	X =  165.960  mm,	Y =   -469.839  mm,	Z =   -309.000  mm,
	W =  90.000 deg,	P =   0.000 deg,	R =   90.000 deg
};
P[3008]{
   GP1:
	UF : 0, UT : 6,		CONFIG : 'N U T, 0, 0, 0',
	X =  164.763  mm,	Y =   -470.352  mm,	Z =   -309.000  mm,
	W =  90.000 deg,	P =   0.000 deg,	R =   90.000 deg
};
P[3009]{
   GP1:
	UF : 0, UT : 6,		CONFIG : 'N U T, 0, 0, 0',
	X =  163.654  mm,	Y =   -470.474  mm,	Z =   -309.000  mm,
	W =  90.000 deg,	P =   0.000 deg,	R =   90.000 deg
};
P[3010]{
   GP1:
	UF : 0, UT : 6,		CONFIG : 'N U T, 0, 0, 0',
	X =  163.001  mm,	Y =   -471.506  mm,	Z =   -309.100  mm,
	W =  90.000 deg,	P =   0.000 deg,	R =   90.000 deg
};
P[3011]{
   GP1:
	UF : 0, UT : 6,		CONFIG : 'N U T, 0, 0, 0',
	X =  162.078  mm,	Y =   -472.109  mm,	Z =   -309.100  mm,
	W =  90.000 deg,	P =   0.000 deg,	R =   90.000 deg
};
P[3012]{
   GP1:
	UF : 0, UT : 6,		CONFIG : 'N U T, 0, 0, 0',
	X =  161.118  mm,	Y =   -472.310  mm,	Z =   -309.000  mm,
	W =  90.000 deg,	P =   0.000 deg,	R =   90.000 deg
};
P[3013]{
   GP1:
	UF : 0, UT : 6,		CONFIG : 'N U T, 0, 0, 0',
	X =  160.747  mm,	Y =   -473.096  mm,	Z =   -309.000  mm,
	W =  90.000 deg,	P =   0.000 deg,	R =   90.000 deg
};
P[3014]{
   GP1:
	UF : 0, UT : 6,		CONFIG : 'N U T, 0, 0, 0',
	X =  159.614  mm,	Y =   -473.326  mm,	Z =   -312.206  mm,
	W =  90.000 deg,	P =   0.000 deg,	R =   90.000 deg
};
P[3015]{
   GP1:
	UF : 0, UT : 6,		CONFIG : 'N U T, 0, 0, 0',
	X =  158.718  mm,	Y =   -474.116  mm,	Z =   -309.000  mm,
	W =  90.000 deg,	P =   0.000 deg,	R =   90.000 deg
};
P[3016]{
   GP1:
	UF : 0, UT : 6,		CONFIG : 'N U T, 0, 0, 0',
	X =  157.157  mm,	Y =   -474.400  mm,	Z =   -309.000  mm,
	W =  90.000 deg,	P =   0.000 deg,	R =   90.000 deg
};
P[3017]{
   GP1:
	UF : 0, UT : 6,		CONFIG : 'N U T, 0, 0, 0',
	X =  156.715  mm,	Y =   -475.159  mm,	Z =   -320.034  mm,
	W =  90.000 deg,	P =   0.000 deg,	R =   90.000 deg
};
P[3018]{
   GP1:
	UF : 0, UT : 6,		CONFIG : 'N U T, 0, 0, 0',
	X =  155.908  mm,	Y =   -475.336  mm,	Z =   -309.000  mm,
	W =  90.000 deg,	P =   0.000 deg,	R =   90.000 deg
};
P[3019]{
   GP1:
	UF : 0, UT : 6,		CONFIG : 'N U T, 0, 0, 0',
	X =  154.941  mm,	Y =   -475.565  mm,	Z =   -309.000  mm,
	W =  90.000 deg,	P =   0.000 deg,	R =   90.000 deg
};
P[3020]{
   GP1:
	UF : 0, UT : 6,		CONFIG : 'N U T, 0, 0, 0',
	X =  154.314  mm,	Y =   -476.515  mm,	Z =   -309.000  mm,
	W =  90.000 deg,	P =   0.000 deg,	R =   90.000 deg
};
P[3021]{
   GP1:
	UF : 0, UT : 6,		CONFIG : 'N U T, 0, 0, 0',
	X =  153.381  mm,	Y =   -476.773  mm,	Z =   -309.000  mm,
	W =  90.000 deg,	P =   0.000 deg,	R =   90.000 deg
};
P[3022]{
   GP1:
	UF : 0, UT : 6,		CONFIG : 'N U T, 0, 0, 0',
	X =  161.189  mm,	Y =   -489.706  mm,	Z =   -309.000  mm,
	W =  90.000 deg,	P =   0.000 deg,	R =   90.000 deg
};
P[3023]{
   GP1:
	UF : 0, UT : 6,		CONFIG : 'N U T, 0, 0, 0',
	X =  162.232  mm,	Y =   -489.306  mm,	Z =   -309.000  mm,
	W =  90.000 deg,	P =   0.000 deg,	R =   90.000 deg
};
P[3024]{
   GP1:
	UF : 0, UT : 6,		CONFIG : 'N U T, 0, 0, 0',
	X =  162.974  mm,	Y =   -488.936  mm,	Z =   -309.000  mm,
	W =  90.000 deg,	P =   0.000 deg,	R =   90.000 deg
};
P[3025]{
   GP1:
	UF : 0, UT : 6,		CONFIG : 'N U T, 0, 0, 0',
	X =  164.233  mm,	Y =   -488.251  mm,	Z =   -309.000  mm,
	W =  90.000 deg,	P =   0.000 deg,	R =   90.000 deg
};
P[3026]{
   GP1:
	UF : 0, UT : 6,		CONFIG : 'N U T, 0, 0, 0',
	X =  166.230  mm,	Y =   -486.702  mm,	Z =   -309.000  mm,
	W =  90.000 deg,	P =   0.000 deg,	R =   90.000 deg
};
P[3027]{
   GP1:
	UF : 0, UT : 6,		CONFIG : 'N U T, 0, 0, 0',
	X =  167.168  mm,	Y =   -486.317  mm,	Z =   -309.000  mm,
	W =  90.000 deg,	P =   0.000 deg,	R =   90.000 deg
};
P[3028]{
   GP1:
	UF : 0, UT : 6,		CONFIG : 'N U T, 0, 0, 0',
	X =  167.771  mm,	Y =   -485.802  mm,	Z =   -309.000  mm,
	W =  90.000 deg,	P =   0.000 deg,	R =   90.000 deg
};
P[3029]{
   GP1:
	UF : 0, UT : 6,		CONFIG : 'N U T, 0, 0, 0',
	X =  168.725  mm,	Y =   -485.608  mm,	Z =   -309.000  mm,
	W =  90.000 deg,	P =   0.000 deg,	R =   90.000 deg
};
P[3030]{
   GP1:
	UF : 0, UT : 6,		CONFIG : 'N U T, 0, 0, 0',
	X =  170.097  mm,	Y =   -485.095  mm,	Z =   -309.000  mm,
	W =  90.000 deg,	P =   0.000 deg,	R =   90.000 deg
};
P[3031]{
   GP1:
	UF : 0, UT : 6,		CONFIG : 'N U T, 0, 0, 0',
	X =  171.086  mm,	Y =   -483.830  mm,	Z =   -310.570  mm,
	W =  90.000 deg,	P =   0.000 deg,	R =   90.000 deg
};
P[3032]{
   GP1:
	UF : 0, UT : 6,		CONFIG : 'N U T, 0, 0, 0',
	X =  172.239  mm,	Y =   -483.433  mm,	Z =   -309.100  mm,
	W =  90.000 deg,	P =   0.000 deg,	R =   90.000 deg
};
P[3033]{
   GP1:
	UF : 0, UT : 6,		CONFIG : 'N U T, 0, 0, 0',
	X =  173.577  mm,	Y =   -482.381  mm,	Z =   -309.100  mm,
	W =  90.000 deg,	P =   0.000 deg,	R =   90.000 deg
};
P[3034]{
   GP1:
	UF : 0, UT : 6,		CONFIG : 'N U T, 0, 0, 0',
	X =  174.632  mm,	Y =   -482.143  mm,	Z =   -316.236  mm,
	W =  90.000 deg,	P =   0.000 deg,	R =   90.000 deg
};
P[3035]{
   GP1:
	UF : 0, UT : 6,		CONFIG : 'N U T, 0, 0, 0',
	X =  176.654  mm,	Y =   -480.667  mm,	Z =   -309.100  mm,
	W =  90.000 deg,	P =   0.000 deg,	R =   90.000 deg
};
P[3036]{
   GP1:
	UF : 0, UT : 6,		CONFIG : 'N U T, 0, 0, 0',
	X =  178.148  mm,	Y =   -479.994  mm,	Z =   -309.100  mm,
	W =  90.000 deg,	P =   0.000 deg,	R =   90.000 deg
};
P[3037]{
   GP1:
	UF : 0, UT : 6,		CONFIG : 'N U T, 0, 0, 0',
	X =  179.964  mm,	Y =   -478.828  mm,	Z =   -309.000  mm,
	W =  90.000 deg,	P =   0.000 deg,	R =   90.000 deg
};
P[3038]{
   GP1:
	UF : 0, UT : 6,		CONFIG : 'N U T, 0, 0, 0',
	X =  181.856  mm,	Y =   -477.882  mm,	Z =   -309.000  mm,
	W =  90.000 deg,	P =   0.000 deg,	R =   90.000 deg
};
P[3039]{
   GP1:
	UF : 0, UT : 6,		CONFIG : 'N U T, 0, 0, 0',
	X =  182.674  mm,	Y =   -477.319  mm,	Z =   -309.000  mm,
	W =  90.000 deg,	P =   0.000 deg,	R =   90.000 deg
};
P[3040]{
   GP1:
	UF : 0, UT : 6,		CONFIG : 'N U T, 0, 0, 0',
	X =  183.656  mm,	Y =   -476.853  mm,	Z =   -309.000  mm,
	W =  90.000 deg,	P =   0.000 deg,	R =   90.000 deg
};
P[3041]{
   GP1:
	UF : 0, UT : 6,		CONFIG : 'N U T, 0, 0, 0',
	X =  185.064  mm,	Y =   -475.764  mm,	Z =   -309.100  mm,
	W =  90.000 deg,	P =   0.000 deg,	R =   90.000 deg
};
P[3042]{
   GP1:
	UF : 0, UT : 6,		CONFIG : 'N U T, 0, 0, 0',
	X =  186.024  mm,	Y =   -475.466  mm,	Z =   -309.000  mm,
	W =  90.000 deg,	P =   0.000 deg,	R =   90.000 deg
};
P[3043]{
   GP1:
	UF : 0, UT : 6,		CONFIG : 'N U T, 0, 0, 0',
	X =  186.459  mm,	Y =   -474.881  mm,	Z =   -309.000  mm,
	W =  90.000 deg,	P =   0.000 deg,	R =   90.000 deg
};
P[3044]{
   GP1:
	UF : 0, UT : 6,		CONFIG : 'N U T, 0, 0, 0',
	X =  187.871  mm,	Y =   -474.561  mm,	Z =   -309.000  mm,
	W =  90.000 deg,	P =   0.000 deg,	R =   90.000 deg
};
P[3045]{
   GP1:
	UF : 0, UT : 6,		CONFIG : 'N U T, 0, 0, 0',
	X =  189.558  mm,	Y =   -473.607  mm,	Z =   -309.000  mm,
	W =  90.000 deg,	P =   0.000 deg,	R =   90.000 deg
};
P[3046]{
   GP1:
	UF : 0, UT : 6,		CONFIG : 'N U T, 0, 0, 0',
	X =  190.537  mm,	Y =   -473.179  mm,	Z =   -309.100  mm,
	W =  90.000 deg,	P =   0.000 deg,	R =   90.000 deg
};
P[3047]{
   GP1:
	UF : 0, UT : 6,		CONFIG : 'N U T, 0, 0, 0',
	X =  190.960  mm,	Y =   -472.234  mm,	Z =   -309.000  mm,
	W =  90.000 deg,	P =   0.000 deg,	R =   90.000 deg
};
P[3048]{
   GP1:
	UF : 0, UT : 6,		CONFIG : 'N U T, 0, 0, 0',
	X =  193.639  mm,	Y =   -470.753  mm,	Z =   -309.000  mm,
	W =  90.000 deg,	P =   0.000 deg,	R =   90.000 deg
};
P[3049]{
   GP1:
	UF : 0, UT : 6,		CONFIG : 'N U T, 0, 0, 0',
	X =  195.285  mm,	Y =   -470.166  mm,	Z =   -309.000  mm,
	W =  90.000 deg,	P =   0.000 deg,	R =   90.000 deg
};
P[3050]{
   GP1:
	UF : 0, UT : 6,		CONFIG : 'N U T, 0, 0, 0',
	X =  196.338  mm,	Y =   -469.341  mm,	Z =   -312.108  mm,
	W =  90.000 deg,	P =   0.000 deg,	R =   90.000 deg
};
P[3051]{
   GP1:
	UF : 0, UT : 6,		CONFIG : 'N U T, 0, 0, 0',
	X =  197.381  mm,	Y =   -469.332  mm,	Z =   -326.194  mm,
	W =  90.000 deg,	P =   0.000 deg,	R =   90.000 deg
};
P[3052]{
   GP1:
	UF : 0, UT : 6,		CONFIG : 'N U T, 0, 0, 0',
	X =  197.799  mm,	Y =   -468.667  mm,	Z =   -320.599  mm,
	W =  90.000 deg,	P =   0.000 deg,	R =   90.000 deg
};
P[3053]{
   GP1:
	UF : 0, UT : 6,		CONFIG : 'N U T, 0, 0, 0',
	X =  199.838  mm,	Y =   -467.568  mm,	Z =   -309.000  mm,
	W =  90.000 deg,	P =   0.000 deg,	R =   90.000 deg
};
P[3054]{
   GP1:
	UF : 0, UT : 6,		CONFIG : 'N U T, 0, 0, 0',
	X =  200.850  mm,	Y =   -467.137  mm,	Z =   -309.000  mm,
	W =  90.000 deg,	P =   0.000 deg,	R =   90.000 deg
};
P[3055]{
   GP1:
	UF : 0, UT : 6,		CONFIG : 'N U T, 0, 0, 0',
	X =  201.586  mm,	Y =   -466.595  mm,	Z =   -309.100  mm,
	W =  90.000 deg,	P =   0.000 deg,	R =   90.000 deg
};
P[3056]{
   GP1:
	UF : 0, UT : 6,		CONFIG : 'N U T, 0, 0, 0',
	X =  202.447  mm,	Y =   -466.499  mm,	Z =   -316.149  mm,
	W =  90.000 deg,	P =   0.000 deg,	R =   90.000 deg
};
P[3057]{
   GP1:
	UF : 0, UT : 6,		CONFIG : 'N U T, 0, 0, 0',
	X =  203.353  mm,	Y =   -465.563  mm,	Z =   -319.247  mm,
	W =  90.000 deg,	P =   0.000 deg,	R =   90.000 deg
};
P[3058]{
   GP1:
	UF : 0, UT : 6,		CONFIG : 'N U T, 0, 0, 0',
	X =  204.948  mm,	Y =   -464.262  mm,	Z =   -309.000  mm,
	W =  90.000 deg,	P =   0.000 deg,	R =   90.000 deg
};
P[3059]{
   GP1:
	UF : 0, UT : 6,		CONFIG : 'N U T, 0, 0, 0',
	X =  206.055  mm,	Y =   -463.667  mm,	Z =   -309.000  mm,
	W =  90.000 deg,	P =   0.000 deg,	R =   90.000 deg
};
P[3060]{
   GP1:
	UF : 0, UT : 6,		CONFIG : 'N U T, 0, 0, 0',
	X =  206.857  mm,	Y =   -463.488  mm,	Z =   -309.000  mm,
	W =  90.000 deg,	P =   0.000 deg,	R =   90.000 deg
};
P[3061]{
   GP1:
	UF : 0, UT : 6,		CONFIG : 'N U T, 0, 0, 0',
	X =  207.561  mm,	Y =   -462.861  mm,	Z =   -309.000  mm,
	W =  90.000 deg,	P =   0.000 deg,	R =   90.000 deg
};
P[3062]{
   GP1:
	UF : 0, UT : 6,		CONFIG : 'N U T, 0, 0, 0',
	X =  208.392  mm,	Y =   -462.080  mm,	Z =   -309.100  mm,
	W =  90.000 deg,	P =   0.000 deg,	R =   90.000 deg
};
P[3063]{
   GP1:
	UF : 0, UT : 6,		CONFIG : 'N U T, 0, 0, 0',
	X =  209.725  mm,	Y =   -462.207  mm,	Z =   -324.192  mm,
	W =  90.000 deg,	P =   0.000 deg,	R =   90.000 deg
};
P[3064]{
   GP1:
	UF : 0, UT : 6,		CONFIG : 'N U T, 0, 0, 0',
	X =  210.434  mm,	Y =   -461.339  mm,	Z =   -309.000  mm,
	W =  90.000 deg,	P =   0.000 deg,	R =   90.000 deg
};
P[3065]{
   GP1:
	UF : 0, UT : 6,		CONFIG : 'N U T, 0, 0, 0',
	X =  211.216  mm,	Y =   -460.996  mm,	Z =   -318.087  mm,
	W =  90.000 deg,	P =   0.000 deg,	R =   90.000 deg
};
P[3066]{
   GP1:
	UF : 0, UT : 6,		CONFIG : 'N U T, 0, 0, 0',
	X =  211.856  mm,	Y =   -460.545  mm,	Z =   -309.000  mm,
	W =  90.000 deg,	P =   0.000 deg,	R =   90.000 deg
};
P[3067]{
   GP1:
	UF : 0, UT : 6,		CONFIG : 'N U T, 0, 0, 0',
	X =  213.067  mm,	Y =   -460.370  mm,	Z =   -316.222  mm,
	W =  90.000 deg,	P =   0.000 deg,	R =   90.000 deg
};
P[3068]{
   GP1:
	UF : 0, UT : 6,		CONFIG : 'N U T, 0, 0, 0',
	X =  213.309  mm,	Y =   -459.472  mm,	Z =   -309.100  mm,
	W =  90.000 deg,	P =   0.000 deg,	R =   90.000 deg
};
P[3069]{
   GP1:
	UF : 0, UT : 6,		CONFIG : 'N U T, 0, 0, 0',
	X =  214.258  mm,	Y =   -459.161  mm,	Z =   -323.141  mm,
	W =  90.000 deg,	P =   0.000 deg,	R =   90.000 deg
};
P[3070]{
   GP1:
	UF : 0, UT : 6,		CONFIG : 'N U T, 0, 0, 0',
	X =  215.681  mm,	Y =   -458.097  mm,	Z =   -320.747  mm,
	W =  90.000 deg,	P =   0.000 deg,	R =   90.000 deg
};
P[3071]{
   GP1:
	UF : 0, UT : 6,		CONFIG : 'N U T, 0, 0, 0',
	X =  216.597  mm,	Y =   -458.003  mm,	Z =   -310.970  mm,
	W =  90.000 deg,	P =   0.000 deg,	R =   90.000 deg
};
P[3072]{
   GP1:
	UF : 0, UT : 6,		CONFIG : 'N U T, 0, 0, 0',
	X =  217.463  mm,	Y =   -457.305  mm,	Z =   -319.124  mm,
	W =  90.000 deg,	P =   0.000 deg,	R =   90.000 deg
};
P[3073]{
   GP1:
	UF : 0, UT : 6,		CONFIG : 'N U T, 0, 0, 0',
	X =  218.185  mm,	Y =   -457.117  mm,	Z =   -309.000  mm,
	W =  90.000 deg,	P =   0.000 deg,	R =   90.000 deg
};
P[3074]{
   GP1:
	UF : 0, UT : 6,		CONFIG : 'N U T, 0, 0, 0',
	X =  219.140  mm,	Y =   -456.645  mm,	Z =   -319.283  mm,
	W =  90.000 deg,	P =   0.000 deg,	R =   90.000 deg
};
P[3075]{
   GP1:
	UF : 0, UT : 6,		CONFIG : 'N U T, 0, 0, 0',
	X =  219.698  mm,	Y =   -456.066  mm,	Z =   -309.000  mm,
	W =  90.000 deg,	P =   0.000 deg,	R =   90.000 deg
};
P[3076]{
   GP1:
	UF : 0, UT : 6,		CONFIG : 'N U T, 0, 0, 0',
	X =  220.893  mm,	Y =   -455.735  mm,	Z =   -325.142  mm,
	W =  90.000 deg,	P =   0.000 deg,	R =   90.000 deg
};
P[3077]{
   GP1:
	UF : 0, UT : 6,		CONFIG : 'N U T, 0, 0, 0',
	X =  221.443  mm,	Y =   -454.761  mm,	Z =   -309.000  mm,
	W =  90.000 deg,	P =   0.000 deg,	R =   90.000 deg
};
P[3078]{
   GP1:
	UF : 0, UT : 6,		CONFIG : 'N U T, 0, 0, 0',
	X =  222.869  mm,	Y =   -454.133  mm,	Z =   -309.000  mm,
	W =  90.000 deg,	P =   0.000 deg,	R =   90.000 deg
};
P[3079]{
   GP1:
	UF : 0, UT : 6,		CONFIG : 'N U T, 0, 0, 0',
	X =  223.946  mm,	Y =   -453.384  mm,	Z =   -309.000  mm,
	W =  90.000 deg,	P =   0.000 deg,	R =   90.000 deg
};
P[3080]{
   GP1:
	UF : 0, UT : 6,		CONFIG : 'N U T, 0, 0, 0',
	X =  225.188  mm,	Y =   -452.814  mm,	Z =   -309.100  mm,
	W =  90.000 deg,	P =   0.000 deg,	R =   90.000 deg
};
P[3081]{
   GP1:
	UF : 0, UT : 6,		CONFIG : 'N U T, 0, 0, 0',
	X =  226.063  mm,	Y =   -452.342  mm,	Z =   -309.000  mm,
	W =  90.000 deg,	P =   0.000 deg,	R =   90.000 deg
};
P[3082]{
   GP1:
	UF : 0, UT : 6,		CONFIG : 'N U T, 0, 0, 0',
	X =  227.719  mm,	Y =   -451.530  mm,	Z =   -309.000  mm,
	W =  90.000 deg,	P =   0.000 deg,	R =   90.000 deg
};
P[3083]{
   GP1:
	UF : 0, UT : 6,		CONFIG : 'N U T, 0, 0, 0',
	X =  228.471  mm,	Y =   -451.139  mm,	Z =   -309.100  mm,
	W =  90.000 deg,	P =   0.000 deg,	R =   90.000 deg
};
P[3084]{
   GP1:
	UF : 0, UT : 6,		CONFIG : 'N U T, 0, 0, 0',
	X =  229.322  mm,	Y =   -450.263  mm,	Z =   -309.100  mm,
	W =  90.000 deg,	P =   0.000 deg,	R =   90.000 deg
};
P[3085]{
   GP1:
	UF : 0, UT : 6,		CONFIG : 'N U T, 0, 0, 0',
	X =  230.058  mm,	Y =   -450.049  mm,	Z =   -309.100  mm,
	W =  90.000 deg,	P =   0.000 deg,	R =   90.000 deg
};
P[3086]{
   GP1:
	UF : 0, UT : 6,		CONFIG : 'N U T, 0, 0, 0',
	X =  231.335  mm,	Y =   -449.319  mm,	Z =   -309.100  mm,
	W =  90.000 deg,	P =   0.000 deg,	R =   90.000 deg
};
P[3087]{
   GP1:
	UF : 0, UT : 6,		CONFIG : 'N U T, 0, 0, 0',
	X =  232.003  mm,	Y =   -448.940  mm,	Z =   -309.000  mm,
	W =  90.000 deg,	P =   0.000 deg,	R =   90.000 deg
};
P[3088]{
   GP1:
	UF : 0, UT : 6,		CONFIG : 'N U T, 0, 0, 0',
	X =  233.065  mm,	Y =   -448.329  mm,	Z =   -309.000  mm,
	W =  90.000 deg,	P =   0.000 deg,	R =   90.000 deg
};
P[3089]{
   GP1:
	UF : 0, UT : 6,		CONFIG : 'N U T, 0, 0, 0',
	X =  234.366  mm,	Y =   -447.530  mm,	Z =   -309.000  mm,
	W =  90.000 deg,	P =   0.000 deg,	R =   90.000 deg
};
P[3090]{
   GP1:
	UF : 0, UT : 6,		CONFIG : 'N U T, 0, 0, 0',
	X =  235.449  mm,	Y =   -446.817  mm,	Z =   -309.000  mm,
	W =  90.000 deg,	P =   0.000 deg,	R =   90.000 deg
};
P[3091]{
   GP1:
	UF : 0, UT : 6,		CONFIG : 'N U T, 0, 0, 0',
	X =  237.066  mm,	Y =   -446.066  mm,	Z =   -309.000  mm,
	W =  90.000 deg,	P =   0.000 deg,	R =   90.000 deg
};
P[3092]{
   GP1:
	UF : 0, UT : 6,		CONFIG : 'N U T, 0, 0, 0',
	X =  237.996  mm,	Y =   -445.243  mm,	Z =   -309.100  mm,
	W =  90.000 deg,	P =   0.000 deg,	R =   90.000 deg
};
P[3093]{
   GP1:
	UF : 0, UT : 6,		CONFIG : 'N U T, 0, 0, 0',
	X =  239.589  mm,	Y =   -444.449  mm,	Z =   -309.000  mm,
	W =  90.000 deg,	P =   0.000 deg,	R =   90.000 deg
};
P[3094]{
   GP1:
	UF : 0, UT : 6,		CONFIG : 'N U T, 0, 0, 0',
	X =  240.520  mm,	Y =   -443.817  mm,	Z =   -309.100  mm,
	W =  90.000 deg,	P =   0.000 deg,	R =   90.000 deg
};
P[3095]{
   GP1:
	UF : 0, UT : 6,		CONFIG : 'N U T, 0, 0, 0',
	X =  241.814  mm,	Y =   -443.197  mm,	Z =   -309.000  mm,
	W =  90.000 deg,	P =   0.000 deg,	R =   90.000 deg
};
P[3096]{
   GP1:
	UF : 0, UT : 6,		CONFIG : 'N U T, 0, 0, 0',
	X =  242.713  mm,	Y =   -442.766  mm,	Z =   -309.100  mm,
	W =  90.000 deg,	P =   0.000 deg,	R =   90.000 deg
};
P[3097]{
   GP1:
	UF : 0, UT : 6,		CONFIG : 'N U T, 0, 0, 0',
	X =  244.190  mm,	Y =   -441.863  mm,	Z =   -309.000  mm,
	W =  90.000 deg,	P =   0.000 deg,	R =   90.000 deg
};
P[3098]{
   GP1:
	UF : 0, UT : 6,		CONFIG : 'N U T, 0, 0, 0',
	X =  245.074  mm,	Y =   -441.722  mm,	Z =   -309.000  mm,
	W =  90.000 deg,	P =   0.000 deg,	R =   90.000 deg
};
P[3099]{
   GP1:
	UF : 0, UT : 6,		CONFIG : 'N U T, 0, 0, 0',
	X =  245.736  mm,	Y =   -441.083  mm,	Z =   -309.000  mm,
	W =  90.000 deg,	P =   0.000 deg,	R =   90.000 deg
};
P[3100]{
   GP1:
	UF : 0, UT : 6,		CONFIG : 'N U T, 0, 0, 0',
	X =  246.253  mm,	Y =   -440.457  mm,	Z =   -327.144  mm,
	W =  90.000 deg,	P =   0.000 deg,	R =   90.000 deg
};
P[3101]{
   GP1:
	UF : 0, UT : 6,		CONFIG : 'N U T, 0, 0, 0',
	X =  247.353  mm,	Y =   -440.603  mm,	Z =   -309.000  mm,
	W =  90.000 deg,	P =   0.000 deg,	R =   90.000 deg
};
P[3102]{
   GP1:
	UF : 0, UT : 6,		CONFIG : 'N U T, 0, 0, 0',
	X =  248.262  mm,	Y =   -439.339  mm,	Z =   -309.000  mm,
	W =  90.000 deg,	P =   0.000 deg,	R =   90.000 deg
};
P[3103]{
   GP1:
	UF : 0, UT : 6,		CONFIG : 'N U T, 0, 0, 0',
	X =  249.447  mm,	Y =   -438.720  mm,	Z =   -311.305  mm,
	W =  90.000 deg,	P =   0.000 deg,	R =   90.000 deg
};
P[3104]{
   GP1:
	UF : 0, UT : 6,		CONFIG : 'N U T, 0, 0, 0',
	X =  249.968  mm,	Y =   -438.198  mm,	Z =   -309.000  mm,
	W =  90.000 deg,	P =   0.000 deg,	R =   90.000 deg
};
P[3105]{
   GP1:
	UF : 0, UT : 6,		CONFIG : 'N U T, 0, 0, 0',
	X =  250.759  mm,	Y =   -437.823  mm,	Z =   -309.000  mm,
	W =  90.000 deg,	P =   0.000 deg,	R =   90.000 deg
};
P[3106]{
   GP1:
	UF : 0, UT : 6,		CONFIG : 'N U T, 0, 0, 0',
	X =  251.597  mm,	Y =   -437.468  mm,	Z =   -309.000  mm,
	W =  90.000 deg,	P =   0.000 deg,	R =   90.000 deg
};
P[3107]{
   GP1:
	UF : 0, UT : 6,		CONFIG : 'N U T, 0, 0, 0',
	X =  252.430  mm,	Y =   -436.757  mm,	Z =   -309.100  mm,
	W =  90.000 deg,	P =   0.000 deg,	R =   90.000 deg
};
P[3108]{
   GP1:
	UF : 0, UT : 6,		CONFIG : 'N U T, 0, 0, 0',
	X =  254.468  mm,	Y =   -436.321  mm,	Z =   -323.840  mm,
	W =  90.000 deg,	P =   0.000 deg,	R =   90.000 deg
};
P[3109]{
   GP1:
	UF : 0, UT : 6,		CONFIG : 'N U T, 0, 0, 0',
	X =  256.029  mm,	Y =   -435.170  mm,	Z =   -311.041  mm,
	W =  90.000 deg,	P =   0.000 deg,	R =   90.000 deg
};
P[3110]{
   GP1:
	UF : 0, UT : 6,		CONFIG : 'N U T, 0, 0, 0',
	X =  257.288  mm,	Y =   -434.608  mm,	Z =   -309.000  mm,
	W =  90.000 deg,	P =   0.000 deg,	R =   90.000 deg
};
P[3111]{
   GP1:
	UF : 0, UT : 6,		CONFIG : 'N U T, 0, 0, 0',
	X =  258.792  mm,	Y =   -433.675  mm,	Z =   -309.000  mm,
	W =  90.000 deg,	P =   0.000 deg,	R =   90.000 deg
};
P[3112]{
   GP1:
	UF : 0, UT : 6,		CONFIG : 'N U T, 0, 0, 0',
	X =  259.578  mm,	Y =   -432.478  mm,	Z =   -309.000  mm,
	W =  90.000 deg,	P =   0.000 deg,	R =   90.000 deg
};
P[3113]{
   GP1:
	UF : 0, UT : 6,		CONFIG : 'N U T, 0, 0, 0',
	X =  260.631  mm,	Y =   -432.212  mm,	Z =   -309.050  mm,
	W =  90.000 deg,	P =   0.000 deg,	R =   90.000 deg
};
P[3114]{
   GP1:
	UF : 0, UT : 6,		CONFIG : 'N U T, 0, 0, 0',
	X =  262.213  mm,	Y =   -431.382  mm,	Z =   -309.000  mm,
	W =  90.000 deg,	P =   0.000 deg,	R =   90.000 deg
};
P[3115]{
   GP1:
	UF : 0, UT : 6,		CONFIG : 'N U T, 0, 0, 0',
	X =  263.149  mm,	Y =   -431.451  mm,	Z =   -309.100  mm,
	W =  90.000 deg,	P =   0.000 deg,	R =   90.000 deg
};
P[3116]{
   GP1:
	UF : 0, UT : 6,		CONFIG : 'N U T, 0, 0, 0',
	X =  264.028  mm,	Y =   -430.671  mm,	Z =   -309.100  mm,
	W =  90.000 deg,	P =   0.000 deg,	R =   90.000 deg
};
P[3117]{
   GP1:
	UF : 0, UT : 6,		CONFIG : 'N U T, 0, 0, 0',
	X =  264.974  mm,	Y =   -429.997  mm,	Z =   -309.100  mm,
	W =  90.000 deg,	P =   0.000 deg,	R =   90.000 deg
};
P[3118]{
   GP1:
	UF : 0, UT : 6,		CONFIG : 'N U T, 0, 0, 0',
	X =  265.683  mm,	Y =   -429.203  mm,	Z =   -309.000  mm,
	W =  90.000 deg,	P =   0.000 deg,	R =   90.000 deg
};
P[3119]{
   GP1:
	UF : 0, UT : 6,		CONFIG : 'N U T, 0, 0, 0',
	X =  266.507  mm,	Y =   -428.883  mm,	Z =   -309.000  mm,
	W =  90.000 deg,	P =   0.000 deg,	R =   90.000 deg
};
P[3120]{
   GP1:
	UF : 0, UT : 6,		CONFIG : 'N U T, 0, 0, 0',
	X =  266.981  mm,	Y =   -428.166  mm,	Z =   -309.000  mm,
	W =  90.000 deg,	P =   0.000 deg,	R =   90.000 deg
};
P[3121]{
   GP1:
	UF : 0, UT : 6,		CONFIG : 'N U T, 0, 0, 0',
	X =  267.993  mm,	Y =   -427.934  mm,	Z =   -309.000  mm,
	W =  90.000 deg,	P =   0.000 deg,	R =   90.000 deg
};
P[3122]{
   GP1:
	UF : 0, UT : 6,		CONFIG : 'N U T, 0, 0, 0',
	X =  269.454  mm,	Y =   -427.191  mm,	Z =   -309.000  mm,
	W =  90.000 deg,	P =   0.000 deg,	R =   90.000 deg
};
P[3123]{
   GP1:
	UF : 0, UT : 6,		CONFIG : 'N U T, 0, 0, 0',
	X =  270.364  mm,	Y =   -426.904  mm,	Z =   -309.100  mm,
	W =  90.000 deg,	P =   0.000 deg,	R =   90.000 deg
};
P[3124]{
   GP1:
	UF : 0, UT : 6,		CONFIG : 'N U T, 0, 0, 0',
	X =  271.038  mm,	Y =   -426.468  mm,	Z =   -309.000  mm,
	W =  90.000 deg,	P =   0.000 deg,	R =   90.000 deg
};
P[3125]{
   GP1:
	UF : 0, UT : 6,		CONFIG : 'N U T, 0, 0, 0',
	X =  272.037  mm,	Y =   -426.276  mm,	Z =   -309.000  mm,
	W =  90.000 deg,	P =   0.000 deg,	R =   90.000 deg
};
P[3126]{
   GP1:
	UF : 0, UT : 6,		CONFIG : 'N U T, 0, 0, 0',
	X =  272.459  mm,	Y =   -425.643  mm,	Z =   -324.061  mm,
	W =  90.000 deg,	P =   0.000 deg,	R =   90.000 deg
};
P[3127]{
   GP1:
	UF : 0, UT : 6,		CONFIG : 'N U T, 0, 0, 0',
	X =  273.163  mm,	Y =   -425.087  mm,	Z =   -309.000  mm,
	W =  90.000 deg,	P =   0.000 deg,	R =   90.000 deg
};
P[3128]{
   GP1:
	UF : 0, UT : 6,		CONFIG : 'N U T, 0, 0, 0',
	X =  274.713  mm,	Y =   -424.625  mm,	Z =   -322.101  mm,
	W =  90.000 deg,	P =   0.000 deg,	R =   90.000 deg
};
P[3129]{
   GP1:
	UF : 0, UT : 6,		CONFIG : 'N U T, 0, 0, 0',
	X =  275.243  mm,	Y =   -423.859  mm,	Z =   -309.000  mm,
	W =  90.000 deg,	P =   0.000 deg,	R =   90.000 deg
};
P[3130]{
   GP1:
	UF : 0, UT : 6,		CONFIG : 'N U T, 0, 0, 0',
	X =  276.293  mm,	Y =   -423.542  mm,	Z =   -309.000  mm,
	W =  90.000 deg,	P =   0.000 deg,	R =   90.000 deg
};
P[3131]{
   GP1:
	UF : 0, UT : 6,		CONFIG : 'N U T, 0, 0, 0',
	X =  276.935  mm,	Y =   -422.550  mm,	Z =   -309.000  mm,
	W =  90.000 deg,	P =   0.000 deg,	R =   90.000 deg
};
P[3132]{
   GP1:
	UF : 0, UT : 6,		CONFIG : 'N U T, 0, 0, 0',
	X =  277.995  mm,	Y =   -422.566  mm,	Z =   -309.100  mm,
	W =  90.000 deg,	P =   0.000 deg,	R =   90.000 deg
};
P[3133]{
   GP1:
	UF : 0, UT : 6,		CONFIG : 'N U T, 0, 0, 0',
	X =  279.606  mm,	Y =   -421.652  mm,	Z =   -309.100  mm,
	W =  90.000 deg,	P =   0.000 deg,	R =   90.000 deg
};
P[3134]{
   GP1:
	UF : 0, UT : 6,		CONFIG : 'N U T, 0, 0, 0',
	X =  280.174  mm,	Y =   -420.921  mm,	Z =   -309.000  mm,
	W =  90.000 deg,	P =   0.000 deg,	R =   90.000 deg
};
P[3135]{
   GP1:
	UF : 0, UT : 6,		CONFIG : 'N U T, 0, 0, 0',
	X =  280.833  mm,	Y =   -420.302  mm,	Z =   -309.000  mm,
	W =  90.000 deg,	P =   0.000 deg,	R =   90.000 deg
};
P[3136]{
   GP1:
	UF : 0, UT : 6,		CONFIG : 'N U T, 0, 0, 0',
	X =  281.961  mm,	Y =   -420.441  mm,	Z =   -309.000  mm,
	W =  90.000 deg,	P =   0.000 deg,	R =   90.000 deg
};
P[3137]{
   GP1:
	UF : 0, UT : 6,		CONFIG : 'N U T, 0, 0, 0',
	X =  282.907  mm,	Y =   -419.349  mm,	Z =   -309.000  mm,
	W =  90.000 deg,	P =   0.000 deg,	R =   90.000 deg
};
P[3138]{
   GP1:
	UF : 0, UT : 6,		CONFIG : 'N U T, 0, 0, 0',
	X =  284.593  mm,	Y =   -418.931  mm,	Z =   -312.196  mm,
	W =  90.000 deg,	P =   0.000 deg,	R =   90.000 deg
};
P[3139]{
   GP1:
	UF : 0, UT : 6,		CONFIG : 'N U T, 0, 0, 0',
	X =  285.638  mm,	Y =   -417.845  mm,	Z =   -309.000  mm,
	W =  90.000 deg,	P =   0.000 deg,	R =   90.000 deg
};
P[3140]{
   GP1:
	UF : 0, UT : 6,		CONFIG : 'N U T, 0, 0, 0',
	X =  287.168  mm,	Y =   -417.399  mm,	Z =   -309.000  mm,
	W =  90.000 deg,	P =   0.000 deg,	R =   90.000 deg
};
P[3141]{
   GP1:
	UF : 0, UT : 6,		CONFIG : 'N U T, 0, 0, 0',
	X =  288.074  mm,	Y =   -416.654  mm,	Z =   -309.000  mm,
	W =  90.000 deg,	P =   0.000 deg,	R =   90.000 deg
};
P[3142]{
   GP1:
	UF : 0, UT : 6,		CONFIG : 'N U T, 0, 0, 0',
	X =  288.701  mm,	Y =   -416.133  mm,	Z =   -309.000  mm,
	W =  90.000 deg,	P =   0.000 deg,	R =   90.000 deg
};
P[3143]{
   GP1:
	UF : 0, UT : 6,		CONFIG : 'N U T, 0, 0, 0',
	X =  289.901  mm,	Y =   -415.539  mm,	Z =   -309.000  mm,
	W =  90.000 deg,	P =   0.000 deg,	R =   90.000 deg
};
P[3144]{
   GP1:
	UF : 0, UT : 6,		CONFIG : 'N U T, 0, 0, 0',
	X =  290.454  mm,	Y =   -414.690  mm,	Z =   -309.100  mm,
	W =  90.000 deg,	P =   0.000 deg,	R =   90.000 deg
};
P[3145]{
   GP1:
	UF : 0, UT : 6,		CONFIG : 'N U T, 0, 0, 0',
	X =  291.404  mm,	Y =   -414.473  mm,	Z =   -309.000  mm,
	W =  90.000 deg,	P =   0.000 deg,	R =   90.000 deg
};
P[3146]{
   GP1:
	UF : 0, UT : 6,		CONFIG : 'N U T, 0, 0, 0',
	X =  293.101  mm,	Y =   -413.861  mm,	Z =   -309.000  mm,
	W =  90.000 deg,	P =   0.000 deg,	R =   90.000 deg
};
P[3147]{
   GP1:
	UF : 0, UT : 6,		CONFIG : 'N U T, 0, 0, 0',
	X =  294.183  mm,	Y =   -413.332  mm,	Z =   -309.100  mm,
	W =  90.000 deg,	P =   0.000 deg,	R =   90.000 deg
};
P[3148]{
   GP1:
	UF : 0, UT : 6,		CONFIG : 'N U T, 0, 0, 0',
	X =  295.158  mm,	Y =   -412.751  mm,	Z =   -309.000  mm,
	W =  90.000 deg,	P =   0.000 deg,	R =   90.000 deg
};
P[3149]{
   GP1:
	UF : 0, UT : 6,		CONFIG : 'N U T, 0, 0, 0',
	X =  296.044  mm,	Y =   -412.164  mm,	Z =   -309.000  mm,
	W =  90.000 deg,	P =   0.000 deg,	R =   90.000 deg
};
P[3150]{
   GP1:
	UF : 0, UT : 6,		CONFIG : 'N U T, 0, 0, 0',
	X =  296.655  mm,	Y =   -411.542  mm,	Z =   -309.100  mm,
	W =  90.000 deg,	P =   0.000 deg,	R =   90.000 deg
};
P[3151]{
   GP1:
	UF : 0, UT : 6,		CONFIG : 'N U T, 0, 0, 0',
	X =  297.891  mm,	Y =   -410.789  mm,	Z =   -309.100  mm,
	W =  90.000 deg,	P =   0.000 deg,	R =   90.000 deg
};
P[3152]{
   GP1:
	UF : 0, UT : 6,		CONFIG : 'N U T, 0, 0, 0',
	X =  298.854  mm,	Y =   -410.035  mm,	Z =   -309.000  mm,
	W =  90.000 deg,	P =   0.000 deg,	R =   90.000 deg
};
P[3153]{
   GP1:
	UF : 0, UT : 6,		CONFIG : 'N U T, 0, 0, 0',
	X =  299.668  mm,	Y =   -410.293  mm,	Z =   -309.100  mm,
	W =  90.000 deg,	P =   0.000 deg,	R =   90.000 deg
};
P[3154]{
   GP1:
	UF : 0, UT : 6,		CONFIG : 'N U T, 0, 0, 0',
	X =  299.957  mm,	Y =   -409.372  mm,	Z =   -309.100  mm,
	W =  90.000 deg,	P =   0.000 deg,	R =   90.000 deg
};
P[3155]{
   GP1:
	UF : 0, UT : 6,		CONFIG : 'N U T, 0, 0, 0',
	X =  301.093  mm,	Y =   -408.898  mm,	Z =   -320.865  mm,
	W =  90.000 deg,	P =   0.000 deg,	R =   90.000 deg
};
P[3156]{
   GP1:
	UF : 0, UT : 6,		CONFIG : 'N U T, 0, 0, 0',
	X =  302.572  mm,	Y =   -408.689  mm,	Z =   -309.000  mm,
	W =  90.000 deg,	P =   0.000 deg,	R =   90.000 deg
};
P[3157]{
   GP1:
	UF : 0, UT : 6,		CONFIG : 'N U T, 0, 0, 0',
	X =  302.970  mm,	Y =   -407.626  mm,	Z =   -309.000  mm,
	W =  90.000 deg,	P =   0.000 deg,	R =   90.000 deg
};
P[3158]{
   GP1:
	UF : 0, UT : 6,		CONFIG : 'N U T, 0, 0, 0',
	X =  303.741  mm,	Y =   -407.135  mm,	Z =   -309.000  mm,
	W =  90.000 deg,	P =   0.000 deg,	R =   90.000 deg
};
P[3159]{
   GP1:
	UF : 0, UT : 6,		CONFIG : 'N U T, 0, 0, 0',
	X =  304.855  mm,	Y =   -407.262  mm,	Z =   -309.100  mm,
	W =  90.000 deg,	P =   0.000 deg,	R =   90.000 deg
};
P[3160]{
   GP1:
	UF : 0, UT : 6,		CONFIG : 'N U T, 0, 0, 0',
	X =  305.478  mm,	Y =   -406.488  mm,	Z =   -309.000  mm,
	W =  90.000 deg,	P =   0.000 deg,	R =   90.000 deg
};
P[3161]{
   GP1:
	UF : 0, UT : 6,		CONFIG : 'N U T, 0, 0, 0',
	X =  307.123  mm,	Y =   -406.045  mm,	Z =   -309.100  mm,
	W =  90.000 deg,	P =   0.000 deg,	R =   90.000 deg
};
P[3162]{
   GP1:
	UF : 0, UT : 6,		CONFIG : 'N U T, 0, 0, 0',
	X =  307.854  mm,	Y =   -404.826  mm,	Z =   -309.033  mm,
	W =  90.000 deg,	P =   0.000 deg,	R =   90.000 deg
};
P[3163]{
   GP1:
	UF : 0, UT : 6,		CONFIG : 'N U T, 0, 0, 0',
	X =  309.131  mm,	Y =   -404.784  mm,	Z =   -309.100  mm,
	W =  90.000 deg,	P =   0.000 deg,	R =   90.000 deg
};
P[3164]{
   GP1:
	UF : 0, UT : 6,		CONFIG : 'N U T, 0, 0, 0',
	X =  309.845  mm,	Y =   -403.952  mm,	Z =   -309.100  mm,
	W =  90.000 deg,	P =   0.000 deg,	R =   90.000 deg
};
P[3165]{
   GP1:
	UF : 0, UT : 6,		CONFIG : 'N U T, 0, 0, 0',
	X =  310.858  mm,	Y =   -403.152  mm,	Z =   -309.000  mm,
	W =  90.000 deg,	P =   0.000 deg,	R =   90.000 deg
};
P[3166]{
   GP1:
	UF : 0, UT : 6,		CONFIG : 'N U T, 0, 0, 0',
	X =  311.586  mm,	Y =   -402.709  mm,	Z =   -309.000  mm,
	W =  90.000 deg,	P =   0.000 deg,	R =   90.000 deg
};
P[3167]{
   GP1:
	UF : 0, UT : 6,		CONFIG : 'N U T, 0, 0, 0',
	X =  312.311  mm,	Y =   -402.773  mm,	Z =   -309.000  mm,
	W =  90.000 deg,	P =   0.000 deg,	R =   90.000 deg
};
P[3168]{
   GP1:
	UF : 0, UT : 6,		CONFIG : 'N U T, 0, 0, 0',
	X =  313.053  mm,	Y =   -402.323  mm,	Z =   -309.100  mm,
	W =  90.000 deg,	P =   0.000 deg,	R =   90.000 deg
};
P[3169]{
   GP1:
	UF : 0, UT : 6,		CONFIG : 'N U T, 0, 0, 0',
	X =  314.188  mm,	Y =   -401.842  mm,	Z =   -309.100  mm,
	W =  90.000 deg,	P =   0.000 deg,	R =   90.000 deg
};
P[3170]{
   GP1:
	UF : 0, UT : 6,		CONFIG : 'N U T, 0, 0, 0',
	X =  314.964  mm,	Y =   -400.864  mm,	Z =   -309.000  mm,
	W =  90.000 deg,	P =   0.000 deg,	R =   90.000 deg
};
P[3171]{
   GP1:
	UF : 0, UT : 6,		CONFIG : 'N U T, 0, 0, 0',
	X =  315.588  mm,	Y =   -400.313  mm,	Z =   -309.000  mm,
	W =  90.000 deg,	P =   0.000 deg,	R =   90.000 deg
};
P[3172]{
   GP1:
	UF : 0, UT : 6,		CONFIG : 'N U T, 0, 0, 0',
	X =  316.389  mm,	Y =   -400.210  mm,	Z =   -309.000  mm,
	W =  90.000 deg,	P =   0.000 deg,	R =   90.000 deg
};
P[3173]{
   GP1:
	UF : 0, UT : 6,		CONFIG : 'N U T, 0, 0, 0',
	X =  317.487  mm,	Y =   -399.398  mm,	Z =   -309.000  mm,
	W =  90.000 deg,	P =   0.000 deg,	R =   90.000 deg
};
P[3174]{
   GP1:
	UF : 0, UT : 6,		CONFIG : 'N U T, 0, 0, 0',
	X =  318.789  mm,	Y =   -399.323  mm,	Z =   -309.000  mm,
	W =  90.000 deg,	P =   0.000 deg,	R =   90.000 deg
};
P[3175]{
   GP1:
	UF : 0, UT : 6,		CONFIG : 'N U T, 0, 0, 0',
	X =  318.884  mm,	Y =   -398.301  mm,	Z =   -309.000  mm,
	W =  90.000 deg,	P =   0.000 deg,	R =   90.000 deg
};
P[3176]{
   GP1:
	UF : 0, UT : 6,		CONFIG : 'N U T, 0, 0, 0',
	X =  320.086  mm,	Y =   -397.948  mm,	Z =   -309.000  mm,
	W =  90.000 deg,	P =   0.000 deg,	R =   90.000 deg
};
P[3177]{
   GP1:
	UF : 0, UT : 6,		CONFIG : 'N U T, 0, 0, 0',
	X =  321.476  mm,	Y =   -397.313  mm,	Z =   -309.100  mm,
	W =  90.000 deg,	P =   0.000 deg,	R =   90.000 deg
};
P[3178]{
   GP1:
	UF : 0, UT : 6,		CONFIG : 'N U T, 0, 0, 0',
	X =  323.081  mm,	Y =   -396.481  mm,	Z =   -309.000  mm,
	W =  90.000 deg,	P =   0.000 deg,	R =   90.000 deg
};
P[3179]{
   GP1:
	UF : 0, UT : 6,		CONFIG : 'N U T, 0, 0, 0',
	X =  324.212  mm,	Y =   -396.058  mm,	Z =   -309.100  mm,
	W =  90.000 deg,	P =   0.000 deg,	R =   90.000 deg
};
P[3180]{
   GP1:
	UF : 0, UT : 6,		CONFIG : 'N U T, 0, 0, 0',
	X =  324.493  mm,	Y =   -394.963  mm,	Z =   -309.100  mm,
	W =  90.000 deg,	P =   0.000 deg,	R =   90.000 deg
};
P[3181]{
   GP1:
	UF : 0, UT : 6,		CONFIG : 'N U T, 0, 0, 0',
	X =  325.264  mm,	Y =   -394.945  mm,	Z =   -309.100  mm,
	W =  90.000 deg,	P =   0.000 deg,	R =   90.000 deg
};
P[3182]{
   GP1:
	UF : 0, UT : 6,		CONFIG : 'N U T, 0, 0, 0',
	X =  326.233  mm,	Y =   -394.283  mm,	Z =   -309.100  mm,
	W =  90.000 deg,	P =   0.000 deg,	R =   90.000 deg
};
P[3183]{
   GP1:
	UF : 0, UT : 6,		CONFIG : 'N U T, 0, 0, 0',
	X =  327.626  mm,	Y =   -393.768  mm,	Z =   -309.000  mm,
	W =  90.000 deg,	P =   0.000 deg,	R =   90.000 deg
};
P[3184]{
   GP1:
	UF : 0, UT : 6,		CONFIG : 'N U T, 0, 0, 0',
	X =  329.137  mm,	Y =   -393.229  mm,	Z =   -309.000  mm,
	W =  90.000 deg,	P =   0.000 deg,	R =   90.000 deg
};
P[3185]{
   GP1:
	UF : 0, UT : 6,		CONFIG : 'N U T, 0, 0, 0',
	X =  329.591  mm,	Y =   -392.364  mm,	Z =   -309.000  mm,
	W =  90.000 deg,	P =   0.000 deg,	R =   90.000 deg
};
P[3186]{
   GP1:
	UF : 0, UT : 6,		CONFIG : 'N U T, 0, 0, 0',
	X =  330.664  mm,	Y =   -391.632  mm,	Z =   -309.000  mm,
	W =  90.000 deg,	P =   0.000 deg,	R =   90.000 deg
};
P[3187]{
   GP1:
	UF : 0, UT : 6,		CONFIG : 'N U T, 0, 0, 0',
	X =  331.564  mm,	Y =   -391.624  mm,	Z =   -309.000  mm,
	W =  90.000 deg,	P =   0.000 deg,	R =   90.000 deg
};
P[3188]{
   GP1:
	UF : 0, UT : 6,		CONFIG : 'N U T, 0, 0, 0',
	X =  332.310  mm,	Y =   -390.786  mm,	Z =   -325.993  mm,
	W =  90.000 deg,	P =   0.000 deg,	R =   90.000 deg
};
P[3189]{
   GP1:
	UF : 0, UT : 6,		CONFIG : 'N U T, 0, 0, 0',
	X =  333.203  mm,	Y =   -390.899  mm,	Z =   -309.000  mm,
	W =  90.000 deg,	P =   0.000 deg,	R =   90.000 deg
};
P[3190]{
   GP1:
	UF : 0, UT : 6,		CONFIG : 'N U T, 0, 0, 0',
	X =  333.996  mm,	Y =   -390.169  mm,	Z =   -309.000  mm,
	W =  90.000 deg,	P =   0.000 deg,	R =   90.000 deg
};
P[3191]{
   GP1:
	UF : 0, UT : 6,		CONFIG : 'N U T, 0, 0, 0',
	X =  341.415  mm,	Y =   -403.266  mm,	Z =   -309.100  mm,
	W =  90.000 deg,	P =   0.000 deg,	R =   90.000 deg
};
P[3192]{
   GP1:
	UF : 0, UT : 6,		CONFIG : 'N U T, 0, 0, 0',
	X =  340.535  mm,	Y =   -403.069  mm,	Z =   -309.000  mm,
	W =  90.000 deg,	P =   0.000 deg,	R =   90.000 deg
};
P[3193]{
   GP1:
	UF : 0, UT : 6,		CONFIG : 'N U T, 0, 0, 0',
	X =  340.148  mm,	Y =   -403.881  mm,	Z =   -309.000  mm,
	W =  90.000 deg,	P =   0.000 deg,	R =   90.000 deg
};
P[3194]{
   GP1:
	UF : 0, UT : 6,		CONFIG : 'N U T, 0, 0, 0',
	X =  339.227  mm,	Y =   -404.232  mm,	Z =   -309.000  mm,
	W =  90.000 deg,	P =   0.000 deg,	R =   90.000 deg
};
P[3195]{
   GP1:
	UF : 0, UT : 6,		CONFIG : 'N U T, 0, 0, 0',
	X =  338.194  mm,	Y =   -404.645  mm,	Z =   -311.898  mm,
	W =  90.000 deg,	P =   0.000 deg,	R =   90.000 deg
};
P[3196]{
   GP1:
	UF : 0, UT : 6,		CONFIG : 'N U T, 0, 0, 0',
	X =  337.156  mm,	Y =   -405.173  mm,	Z =   -309.100  mm,
	W =  90.000 deg,	P =   0.000 deg,	R =   90.000 deg
};
P[3197]{
   GP1:
	UF : 0, UT : 6,		CONFIG : 'N U T, 0, 0, 0',
	X =  335.370  mm,	Y =   -406.482  mm,	Z =   -309.000  mm,
	W =  90.000 deg,	P =   0.000 deg,	R =   90.000 deg
};
P[3198]{
   GP1:
	UF : 0, UT : 6,		CONFIG : 'N U T, 0, 0, 0',
	X =  334.478  mm,	Y =   -407.273  mm,	Z =   -309.100  mm,
	W =  90.000 deg,	P =   0.000 deg,	R =   90.000 deg
};
P[3199]{
   GP1:
	UF : 0, UT : 6,		CONFIG : 'N U T, 0, 0, 0',
	X =  333.604  mm,	Y =   -407.675  mm,	Z =   -309.000  mm,
	W =  90.000 deg,	P =   0.000 deg,	R =   90.000 deg
};
P[3200]{
   GP1:
	UF : 0, UT : 6,		CONFIG : 'N U T, 0, 0, 0',
	X =  332.753  mm,	Y =   -407.650  mm,	Z =   -309.000  mm,
	W =  90.000 deg,	P =   0.000 deg,	R =   90.000 deg
};
P[3201]{
   GP1:
	UF : 0, UT : 6,		CONFIG : 'N U T, 0, 0, 0',
	X =  331.874  mm,	Y =   -408.861  mm,	Z =   -309.100  mm,
	W =  90.000 deg,	P =   0.000 deg,	R =   90.000 deg
};
P[3202]{
   GP1:
	UF : 0, UT : 6,		CONFIG : 'N U T, 0, 0, 0',
	X =  331.186  mm,	Y =   -409.115  mm,	Z =   -309.000  mm,
	W =  90.000 deg,	P =   0.000 deg,	R =   90.000 deg
};
P[3203]{
   GP1:
	UF : 0, UT : 6,		CONFIG : 'N U T, 0, 0, 0',
	X =  330.283  mm,	Y =   -409.596  mm,	Z =   -309.100  mm,
	W =  90.000 deg,	P =   0.000 deg,	R =   90.000 deg
};
P[3204]{
   GP1:
	UF : 0, UT : 6,		CONFIG : 'N U T, 0, 0, 0',
	X =  329.083  mm,	Y =   -409.874  mm,	Z =   -315.562  mm,
	W =  90.000 deg,	P =   0.000 deg,	R =   90.000 deg
};
P[3205]{
   GP1:
	UF : 0, UT : 6,		CONFIG : 'N U T, 0, 0, 0',
	X =  327.493  mm,	Y =   -411.124  mm,	Z =   -309.000  mm,
	W =  90.000 deg,	P =   0.000 deg,	R =   90.000 deg
};
P[3206]{
   GP1:
	UF : 0, UT : 6,		CONFIG : 'N U T, 0, 0, 0',
	X =  326.758  mm,	Y =   -411.333  mm,	Z =   -309.000  mm,
	W =  90.000 deg,	P =   0.000 deg,	R =   90.000 deg
};
P[3207]{
   GP1:
	UF : 0, UT : 6,		CONFIG : 'N U T, 0, 0, 0',
	X =  326.458  mm,	Y =   -412.093  mm,	Z =   -309.000  mm,
	W =  90.000 deg,	P =   0.000 deg,	R =   90.000 deg
};
P[3208]{
   GP1:
	UF : 0, UT : 6,		CONFIG : 'N U T, 0, 0, 0',
	X =  325.294  mm,	Y =   -412.080  mm,	Z =   -309.000  mm,
	W =  90.000 deg,	P =   0.000 deg,	R =   90.000 deg
};
P[3209]{
   GP1:
	UF : 0, UT : 6,		CONFIG : 'N U T, 0, 0, 0',
	X =  324.335  mm,	Y =   -412.714  mm,	Z =   -309.000  mm,
	W =  90.000 deg,	P =   0.000 deg,	R =   90.000 deg
};
P[3210]{
   GP1:
	UF : 0, UT : 6,		CONFIG : 'N U T, 0, 0, 0',
	X =  323.397  mm,	Y =   -413.417  mm,	Z =   -309.100  mm,
	W =  90.000 deg,	P =   0.000 deg,	R =   90.000 deg
};
P[3211]{
   GP1:
	UF : 0, UT : 6,		CONFIG : 'N U T, 0, 0, 0',
	X =  322.140  mm,	Y =   -413.712  mm,	Z =   -309.000  mm,
	W =  90.000 deg,	P =   0.000 deg,	R =   90.000 deg
};
P[3212]{
   GP1:
	UF : 0, UT : 6,		CONFIG : 'N U T, 0, 0, 0',
	X =  321.655  mm,	Y =   -414.561  mm,	Z =   -309.100  mm,
	W =  90.000 deg,	P =   0.000 deg,	R =   90.000 deg
};
P[3213]{
   GP1:
	UF : 0, UT : 6,		CONFIG : 'N U T, 0, 0, 0',
	X =  321.152  mm,	Y =   -415.123  mm,	Z =   -309.201  mm,
	W =  90.000 deg,	P =   0.000 deg,	R =   90.000 deg
};
P[3214]{
   GP1:
	UF : 0, UT : 6,		CONFIG : 'N U T, 0, 0, 0',
	X =  319.716  mm,	Y =   -415.965  mm,	Z =   -309.000  mm,
	W =  90.000 deg,	P =   0.000 deg,	R =   90.000 deg
};
P[3215]{
   GP1:
	UF : 0, UT : 6,		CONFIG : 'N U T, 0, 0, 0',
	X =  318.873  mm,	Y =   -416.428  mm,	Z =   -309.000  mm,
	W =  90.000 deg,	P =   0.000 deg,	R =   90.000 deg
};
P[3216]{
   GP1:
	UF : 0, UT : 6,		CONFIG : 'N U T, 0, 0, 0',
	X =  317.083  mm,	Y =   -417.008  mm,	Z =   -309.000  mm,
	W =  90.000 deg,	P =   0.000 deg,	R =   90.000 deg
};
P[3217]{
   GP1:
	UF : 0, UT : 6,		CONFIG : 'N U T, 0, 0, 0',
	X =  316.060  mm,	Y =   -417.441  mm,	Z =   -309.100  mm,
	W =  90.000 deg,	P =   0.000 deg,	R =   90.000 deg
};
P[3218]{
   GP1:
	UF : 0, UT : 6,		CONFIG : 'N U T, 0, 0, 0',
	X =  315.602  mm,	Y =   -418.081  mm,	Z =   -309.100  mm,
	W =  90.000 deg,	P =   0.000 deg,	R =   90.000 deg
};
P[3219]{
   GP1:
	UF : 0, UT : 6,		CONFIG : 'N U T, 0, 0, 0',
	X =  314.664  mm,	Y =   -418.077  mm,	Z =   -309.000  mm,
	W =  90.000 deg,	P =   0.000 deg,	R =   90.000 deg
};
P[3220]{
   GP1:
	UF : 0, UT : 6,		CONFIG : 'N U T, 0, 0, 0',
	X =  313.962  mm,	Y =   -418.771  mm,	Z =   -309.000  mm,
	W =  90.000 deg,	P =   0.000 deg,	R =   90.000 deg
};
P[3221]{
   GP1:
	UF : 0, UT : 6,		CONFIG : 'N U T, 0, 0, 0',
	X =  313.017  mm,	Y =   -419.861  mm,	Z =   -311.050  mm,
	W =  90.000 deg,	P =   0.000 deg,	R =   90.000 deg
};
P[3222]{
   GP1:
	UF : 0, UT : 6,		CONFIG : 'N U T, 0, 0, 0',
	X =  312.425  mm,	Y =   -420.081  mm,	Z =   -309.000  mm,
	W =  90.000 deg,	P =   0.000 deg,	R =   90.000 deg
};
P[3223]{
   GP1:
	UF : 0, UT : 6,		CONFIG : 'N U T, 0, 0, 0',
	X =  312.258  mm,	Y =   -419.950  mm,	Z =   -309.100  mm,
	W =  90.000 deg,	P =   0.000 deg,	R =   90.000 deg
};
P[3224]{
   GP1:
	UF : 0, UT : 6,		CONFIG : 'N U T, 0, 0, 0',
	X =  311.923  mm,	Y =   -420.063  mm,	Z =   -309.000  mm,
	W =  90.000 deg,	P =   0.000 deg,	R =   90.000 deg
};
P[3225]{
   GP1:
	UF : 0, UT : 6,		CONFIG : 'N U T, 0, 0, 0',
	X =  311.627  mm,	Y =   -420.173  mm,	Z =   -309.000  mm,
	W =  90.000 deg,	P =   0.000 deg,	R =   90.000 deg
};
P[3226]{
   GP1:
	UF : 0, UT : 6,		CONFIG : 'N U T, 0, 0, 0',
	X =  311.468  mm,	Y =   -420.529  mm,	Z =   -309.100  mm,
	W =  90.000 deg,	P =   0.000 deg,	R =   90.000 deg
};
P[3227]{
   GP1:
	UF : 0, UT : 6,		CONFIG : 'N U T, 0, 0, 0',
	X =  311.355  mm,	Y =   -420.385  mm,	Z =   -309.000  mm,
	W =  90.000 deg,	P =   0.000 deg,	R =   90.000 deg
};
P[3228]{
   GP1:
	UF : 0, UT : 6,		CONFIG : 'N U T, 0, 0, 0',
	X =  311.189  mm,	Y =   -420.110  mm,	Z =   -309.000  mm,
	W =  90.000 deg,	P =   0.000 deg,	R =   90.000 deg
};
P[3229]{
   GP1:
	UF : 0, UT : 6,		CONFIG : 'N U T, 0, 0, 0',
	X =  311.147  mm,	Y =   -420.794  mm,	Z =   -309.100  mm,
	W =  90.000 deg,	P =   0.000 deg,	R =   90.000 deg
};
P[3230]{
   GP1:
	UF : 0, UT : 6,		CONFIG : 'N U T, 0, 0, 0',
	X =  310.746  mm,	Y =   -420.645  mm,	Z =   -309.000  mm,
	W =  90.000 deg,	P =   0.000 deg,	R =   90.000 deg
};
P[3231]{
   GP1:
	UF : 0, UT : 6,		CONFIG : 'N U T, 0, 0, 0',
	X =  310.336  mm,	Y =   -420.960  mm,	Z =   -309.000  mm,
	W =  90.000 deg,	P =   0.000 deg,	R =   90.000 deg
};
P[3232]{
   GP1:
	UF : 0, UT : 6,		CONFIG : 'N U T, 0, 0, 0',
	X =  309.671  mm,	Y =   -421.659  mm,	Z =   -309.100  mm,
	W =  90.000 deg,	P =   0.000 deg,	R =   90.000 deg
};
P[3233]{
   GP1:
	UF : 0, UT : 6,		CONFIG : 'N U T, 0, 0, 0',
	X =  309.509  mm,	Y =   -421.437  mm,	Z =   -309.000  mm,
	W =  90.000 deg,	P =   0.000 deg,	R =   90.000 deg
};
P[3234]{
   GP1:
	UF : 0, UT : 6,		CONFIG : 'N U T, 0, 0, 0',
	X =  309.255  mm,	Y =   -421.209  mm,	Z =   -309.100  mm,
	W =  90.000 deg,	P =   0.000 deg,	R =   90.000 deg
};
P[3235]{
   GP1:
	UF : 0, UT : 6,		CONFIG : 'N U T, 0, 0, 0',
	X =  308.897  mm,	Y =   -421.670  mm,	Z =   -309.100  mm,
	W =  90.000 deg,	P =   0.000 deg,	R =   90.000 deg
};
P[3236]{
   GP1:
	UF : 0, UT : 6,		CONFIG : 'N U T, 0, 0, 0',
	X =  308.705  mm,	Y =   -422.007  mm,	Z =   -309.000  mm,
	W =  90.000 deg,	P =   0.000 deg,	R =   90.000 deg
};
P[3237]{
   GP1:
	UF : 0, UT : 6,		CONFIG : 'N U T, 0, 0, 0',
	X =  308.001  mm,	Y =   -421.834  mm,	Z =   -309.000  mm,
	W =  90.000 deg,	P =   0.000 deg,	R =   90.000 deg
};
P[3238]{
   GP1:
	UF : 0, UT : 6,		CONFIG : 'N U T, 0, 0, 0',
	X =  307.895  mm,	Y =   -422.131  mm,	Z =   -309.000  mm,
	W =  90.000 deg,	P =   0.000 deg,	R =   90.000 deg
};
P[3239]{
   GP1:
	UF : 0, UT : 6,		CONFIG : 'N U T, 0, 0, 0',
	X =  307.925  mm,	Y =   -422.585  mm,	Z =   -312.966  mm,
	W =  90.000 deg,	P =   0.000 deg,	R =   90.000 deg
};
P[3240]{
   GP1:
	UF : 0, UT : 6,		CONFIG : 'N U T, 0, 0, 0',
	X =  306.720  mm,	Y =   -422.838  mm,	Z =   -311.283  mm,
	W =  90.000 deg,	P =   0.000 deg,	R =   90.000 deg
};
P[3241]{
   GP1:
	UF : 0, UT : 6,		CONFIG : 'N U T, 0, 0, 0',
	X =  306.829  mm,	Y =   -423.203  mm,	Z =   -309.000  mm,
	W =  90.000 deg,	P =   0.000 deg,	R =   90.000 deg
};
P[3242]{
   GP1:
	UF : 0, UT : 6,		CONFIG : 'N U T, 0, 0, 0',
	X =  306.035  mm,	Y =   -423.469  mm,	Z =   -309.000  mm,
	W =  90.000 deg,	P =   0.000 deg,	R =   90.000 deg
};
P[3243]{
   GP1:
	UF : 0, UT : 6,		CONFIG : 'N U T, 0, 0, 0',
	X =  305.369  mm,	Y =   -423.315  mm,	Z =   -309.000  mm,
	W =  90.000 deg,	P =   0.000 deg,	R =   90.000 deg
};
P[3244]{
   GP1:
	UF : 0, UT : 6,		CONFIG : 'N U T, 0, 0, 0',
	X =  305.164  mm,	Y =   -423.774  mm,	Z =   -309.000  mm,
	W =  90.000 deg,	P =   0.000 deg,	R =   90.000 deg
};
P[3245]{
   GP1:
	UF : 0, UT : 6,		CONFIG : 'N U T, 0, 0, 0',
	X =  305.121  mm,	Y =   -424.331  mm,	Z =   -309.000  mm,
	W =  90.000 deg,	P =   0.000 deg,	R =   90.000 deg
};
P[3246]{
   GP1:
	UF : 0, UT : 6,		CONFIG : 'N U T, 0, 0, 0',
	X =  304.355  mm,	Y =   -424.020  mm,	Z =   -309.000  mm,
	W =  90.000 deg,	P =   0.000 deg,	R =   90.000 deg
};
P[3247]{
   GP1:
	UF : 0, UT : 6,		CONFIG : 'N U T, 0, 0, 0',
	X =  303.691  mm,	Y =   -424.640  mm,	Z =   -309.000  mm,
	W =  90.000 deg,	P =   0.000 deg,	R =   90.000 deg
};
P[3248]{
   GP1:
	UF : 0, UT : 6,		CONFIG : 'N U T, 0, 0, 0',
	X =  303.482  mm,	Y =   -425.302  mm,	Z =   -309.000  mm,
	W =  90.000 deg,	P =   0.000 deg,	R =   90.000 deg
};
P[3249]{
   GP1:
	UF : 0, UT : 6,		CONFIG : 'N U T, 0, 0, 0',
	X =  302.721  mm,	Y =   -424.951  mm,	Z =   -309.000  mm,
	W =  90.000 deg,	P =   0.000 deg,	R =   90.000 deg
};
P[3250]{
   GP1:
	UF : 0, UT : 6,		CONFIG : 'N U T, 0, 0, 0',
	X =  302.366  mm,	Y =   -425.478  mm,	Z =   -309.000  mm,
	W =  90.000 deg,	P =   0.000 deg,	R =   90.000 deg
};
P[3251]{
   GP1:
	UF : 0, UT : 6,		CONFIG : 'N U T, 0, 0, 0',
	X =  301.574  mm,	Y =   -425.557  mm,	Z =   -311.408  mm,
	W =  90.000 deg,	P =   0.000 deg,	R =   90.000 deg
};
P[3252]{
   GP1:
	UF : 0, UT : 6,		CONFIG : 'N U T, 0, 0, 0',
	X =  301.879  mm,	Y =   -426.423  mm,	Z =   -323.966  mm,
	W =  90.000 deg,	P =   0.000 deg,	R =   90.000 deg
};
P[3253]{
   GP1:
	UF : 0, UT : 6,		CONFIG : 'N U T, 0, 0, 0',
	X =  300.929  mm,	Y =   -426.189  mm,	Z =   -309.000  mm,
	W =  90.000 deg,	P =   0.000 deg,	R =   90.000 deg
};
P[3254]{
   GP1:
	UF : 0, UT : 6,		CONFIG : 'N U T, 0, 0, 0',
	X =  300.366  mm,	Y =   -426.722  mm,	Z =   -309.000  mm,
	W =  90.000 deg,	P =   0.000 deg,	R =   90.000 deg
};
P[3255]{
   GP1:
	UF : 0, UT : 6,		CONFIG : 'N U T, 0, 0, 0',
	X =  300.219  mm,	Y =   -427.294  mm,	Z =   -309.100  mm,
	W =  90.000 deg,	P =   0.000 deg,	R =   90.000 deg
};
P[3256]{
   GP1:
	UF : 0, UT : 6,		CONFIG : 'N U T, 0, 0, 0',
	X =  299.030  mm,	Y =   -427.246  mm,	Z =   -309.000  mm,
	W =  90.000 deg,	P =   0.000 deg,	R =   90.000 deg
};
P[3257]{
   GP1:
	UF : 0, UT : 6,		CONFIG : 'N U T, 0, 0, 0',
	X =  299.241  mm,	Y =   -427.847  mm,	Z =   -309.000  mm,
	W =  90.000 deg,	P =   0.000 deg,	R =   90.000 deg
};
P[3258]{
   GP1:
	UF : 0, UT : 6,		CONFIG : 'N U T, 0, 0, 0',
	X =  298.224  mm,	Y =   -428.041  mm,	Z =   -309.000  mm,
	W =  90.000 deg,	P =   0.000 deg,	R =   90.000 deg
};
P[3259]{
   GP1:
	UF : 0, UT : 6,		CONFIG : 'N U T, 0, 0, 0',
	X =  297.622  mm,	Y =   -428.493  mm,	Z =   -309.000  mm,
	W =  90.000 deg,	P =   0.000 deg,	R =   90.000 deg
};
P[3260]{
   GP1:
	UF : 0, UT : 6,		CONFIG : 'N U T, 0, 0, 0',
	X =  297.292  mm,	Y =   -428.115  mm,	Z =   -309.000  mm,
	W =  90.000 deg,	P =   0.000 deg,	R =   90.000 deg
};
P[3261]{
   GP1:
	UF : 0, UT : 6,		CONFIG : 'N U T, 0, 0, 0',
	X =  296.710  mm,	Y =   -428.809  mm,	Z =   -309.000  mm,
	W =  90.000 deg,	P =   0.000 deg,	R =   90.000 deg
};
P[3262]{
   GP1:
	UF : 0, UT : 6,		CONFIG : 'N U T, 0, 0, 0',
	X =  296.189  mm,	Y =   -429.659  mm,	Z =   -309.100  mm,
	W =  90.000 deg,	P =   0.000 deg,	R =   90.000 deg
};
P[3263]{
   GP1:
	UF : 0, UT : 6,		CONFIG : 'N U T, 0, 0, 0',
	X =  295.396  mm,	Y =   -429.492  mm,	Z =   -309.000  mm,
	W =  90.000 deg,	P =   0.000 deg,	R =   90.000 deg
};
P[3264]{
   GP1:
	UF : 0, UT : 6,		CONFIG : 'N U T, 0, 0, 0',
	X =  295.083  mm,	Y =   -430.354  mm,	Z =   -326.614  mm,
	W =  90.000 deg,	P =   0.000 deg,	R =   90.000 deg
};
P[3265]{
   GP1:
	UF : 0, UT : 6,		CONFIG : 'N U T, 0, 0, 0',
	X =  294.805  mm,	Y =   -429.893  mm,	Z =   -309.000  mm,
	W =  90.000 deg,	P =   0.000 deg,	R =   90.000 deg
};
P[3266]{
   GP1:
	UF : 0, UT : 6,		CONFIG : 'N U T, 0, 0, 0',
	X =  294.444  mm,	Y =   -430.524  mm,	Z =   -309.000  mm,
	W =  90.000 deg,	P =   0.000 deg,	R =   90.000 deg
};
P[3267]{
   GP1:
	UF : 0, UT : 6,		CONFIG : 'N U T, 0, 0, 0',
	X =  293.939  mm,	Y =   -429.903  mm,	Z =   -318.610  mm,
	W =  90.000 deg,	P =   0.000 deg,	R =   90.000 deg
};
P[3268]{
   GP1:
	UF : 0, UT : 6,		CONFIG : 'N U T, 0, 0, 0',
	X =  293.058  mm,	Y =   -430.739  mm,	Z =   -309.100  mm,
	W =  90.000 deg,	P =   0.000 deg,	R =   90.000 deg
};
P[3269]{
   GP1:
	UF : 0, UT : 6,		CONFIG : 'N U T, 0, 0, 0',
	X =  292.275  mm,	Y =   -431.408  mm,	Z =   -309.000  mm,
	W =  90.000 deg,	P =   0.000 deg,	R =   90.000 deg
};
P[3270]{
   GP1:
	UF : 0, UT : 6,		CONFIG : 'N U T, 0, 0, 0',
	X =  291.563  mm,	Y =   -431.913  mm,	Z =   -325.179  mm,
	W =  90.000 deg,	P =   0.000 deg,	R =   90.000 deg
};
P[3271]{
   GP1:
	UF : 0, UT : 6,		CONFIG : 'N U T, 0, 0, 0',
	X =  290.947  mm,	Y =   -431.622  mm,	Z =   -313.218  mm,
	W =  90.000 deg,	P =   0.000 deg,	R =   90.000 deg
};
P[3272]{
   GP1:
	UF : 0, UT : 6,		CONFIG : 'N U T, 0, 0, 0',
	X =  291.001  mm,	Y =   -432.378  mm,	Z =   -309.100  mm,
	W =  90.000 deg,	P =   0.000 deg,	R =   90.000 deg
};
P[3273]{
   GP1:
	UF : 0, UT : 6,		CONFIG : 'N U T, 0, 0, 0',
	X =  290.230  mm,	Y =   -432.329  mm,	Z =   -309.100  mm,
	W =  90.000 deg,	P =   0.000 deg,	R =   90.000 deg
};
P[3274]{
   GP1:
	UF : 0, UT : 6,		CONFIG : 'N U T, 0, 0, 0',
	X =  289.168  mm,	Y =   -433.041  mm,	Z =   -309.100  mm,
	W =  90.000 deg,	P =   0.000 deg,	R =   90.000 deg
};
P[3275]{
   GP1:
	UF : 0, UT : 6,		CONFIG : 'N U T, 0, 0, 0',
	X =  289.330  mm,	Y =   -433.494  mm,	Z =   -309.100  mm,
	W =  90.000 deg,	P =   0.000 deg,	R =   90.000 deg
};
P[3276]{
   GP1:
	UF : 0, UT : 6,		CONFIG : 'N U T, 0, 0, 0',
	X =  288.499  mm,	Y =   -434.024  mm,	Z =   -309.100  mm,
	W =  90.000 deg,	P =   0.000 deg,	R =   90.000 deg
};
P[3277]{
   GP1:
	UF : 0, UT : 6,		CONFIG : 'N U T, 0, 0, 0',
	X =  287.723  mm,	Y =   -433.912  mm,	Z =   -309.000  mm,
	W =  90.000 deg,	P =   0.000 deg,	R =   90.000 deg
};
P[3278]{
   GP1:
	UF : 0, UT : 6,		CONFIG : 'N U T, 0, 0, 0',
	X =  287.164  mm,	Y =   -434.415  mm,	Z =   -317.166  mm,
	W =  90.000 deg,	P =   0.000 deg,	R =   90.000 deg
};
P[3279]{
   GP1:
	UF : 0, UT : 6,		CONFIG : 'N U T, 0, 0, 0',
	X =  286.915  mm,	Y =   -434.047  mm,	Z =   -309.000  mm,
	W =  90.000 deg,	P =   0.000 deg,	R =   90.000 deg
};
P[3280]{
   GP1:
	UF : 0, UT : 6,		CONFIG : 'N U T, 0, 0, 0',
	X =  287.290  mm,	Y =   -434.803  mm,	Z =   -309.000  mm,
	W =  90.000 deg,	P =   0.000 deg,	R =   90.000 deg
};
P[3281]{
   GP1:
	UF : 0, UT : 6,		CONFIG : 'N U T, 0, 0, 0',
	X =  286.421  mm,	Y =   -434.921  mm,	Z =   -309.100  mm,
	W =  90.000 deg,	P =   0.000 deg,	R =   90.000 deg
};
P[3282]{
   GP1:
	UF : 0, UT : 6,		CONFIG : 'N U T, 0, 0, 0',
	X =  285.497  mm,	Y =   -435.166  mm,	Z =   -309.000  mm,
	W =  90.000 deg,	P =   0.000 deg,	R =   90.000 deg
};
P[3283]{
   GP1:
	UF : 0, UT : 6,		CONFIG : 'N U T, 0, 0, 0',
	X =  284.612  mm,	Y =   -435.431  mm,	Z =   -309.000  mm,
	W =  90.000 deg,	P =   0.000 deg,	R =   90.000 deg
};
P[3284]{
   GP1:
	UF : 0, UT : 6,		CONFIG : 'N U T, 0, 0, 0',
	X =  284.588  mm,	Y =   -435.920  mm,	Z =   -309.000  mm,
	W =  90.000 deg,	P =   0.000 deg,	R =   90.000 deg
};
P[3285]{
   GP1:
	UF : 0, UT : 6,		CONFIG : 'N U T, 0, 0, 0',
	X =  284.658  mm,	Y =   -436.283  mm,	Z =   -309.000  mm,
	W =  90.000 deg,	P =   0.000 deg,	R =   90.000 deg
};
P[3286]{
   GP1:
	UF : 0, UT : 6,		CONFIG : 'N U T, 0, 0, 0',
	X =  283.844  mm,	Y =   -436.358  mm,	Z =   -309.000  mm,
	W =  90.000 deg,	P =   0.000 deg,	R =   90.000 deg
};
P[3287]{
   GP1:
	UF : 0, UT : 6,		CONFIG : 'N U T, 0, 0, 0',
	X =  283.502  mm,	Y =   -436.283  mm,	Z =   -315.280  mm,
	W =  90.000 deg,	P =   0.000 deg,	R =   90.000 deg
};
P[3288]{
   GP1:
	UF : 0, UT : 6,		CONFIG : 'N U T, 0, 0, 0',
	X =  282.600  mm,	Y =   -436.649  mm,	Z =   -309.000  mm,
	W =  90.000 deg,	P =   0.000 deg,	R =   90.000 deg
};
P[3289]{
   GP1:
	UF : 0, UT : 6,		CONFIG : 'N U T, 0, 0, 0',
	X =  282.889  mm,	Y =   -437.271  mm,	Z =   -322.368  mm,
	W =  90.000 deg,	P =   0.000 deg,	R =   90.000 deg
};
P[3290]{
   GP1:
	UF : 0, UT : 6,		CONFIG : 'N U T, 0, 0, 0',
	X =  281.986  mm,	Y =   -437.656  mm,	Z =   -309.000  mm,
	W =  90.000 deg,	P =   0.000 deg,	R =   90.000 deg
};
P[3291]{
   GP1:
	UF : 0, UT : 6,		CONFIG : 'N U T, 0, 0, 0',
	X =  281.649  mm,	Y =   -437.301  mm,	Z =   -309.000  mm,
	W =  90.000 deg,	P =   0.000 deg,	R =   90.000 deg
};
P[3292]{
   GP1:
	UF : 0, UT : 6,		CONFIG : 'N U T, 0, 0, 0',
	X =  280.900  mm,	Y =   -437.465  mm,	Z =   -309.000  mm,
	W =  90.000 deg,	P =   0.000 deg,	R =   90.000 deg
};
P[3293]{
   GP1:
	UF : 0, UT : 6,		CONFIG : 'N U T, 0, 0, 0',
	X =  280.488  mm,	Y =   -437.925  mm,	Z =   -316.660  mm,
	W =  90.000 deg,	P =   0.000 deg,	R =   90.000 deg
};
P[3294]{
   GP1:
	UF : 0, UT : 6,		CONFIG : 'N U T, 0, 0, 0',
	X =  280.139  mm,	Y =   -438.378  mm,	Z =   -310.405  mm,
	W =  90.000 deg,	P =   0.000 deg,	R =   90.000 deg
};
P[3295]{
   GP1:
	UF : 0, UT : 6,		CONFIG : 'N U T, 0, 0, 0',
	X =  280.246  mm,	Y =   -438.630  mm,	Z =   -309.100  mm,
	W =  90.000 deg,	P =   0.000 deg,	R =   90.000 deg
};
P[3296]{
   GP1:
	UF : 0, UT : 6,		CONFIG : 'N U T, 0, 0, 0',
	X =  279.931  mm,	Y =   -438.178  mm,	Z =   -309.000  mm,
	W =  90.000 deg,	P =   0.000 deg,	R =   90.000 deg
};
P[3297]{
   GP1:
	UF : 0, UT : 6,		CONFIG : 'N U T, 0, 0, 0',
	X =  279.867  mm,	Y =   -438.067  mm,	Z =   -309.000  mm,
	W =  90.000 deg,	P =   0.000 deg,	R =   90.000 deg
};
P[3298]{
   GP1:
	UF : 0, UT : 6,		CONFIG : 'N U T, 0, 0, 0',
	X =  279.467  mm,	Y =   -438.257  mm,	Z =   -309.100  mm,
	W =  90.000 deg,	P =   0.000 deg,	R =   90.000 deg
};
P[3299]{
   GP1:
	UF : 0, UT : 6,		CONFIG : 'N U T, 0, 0, 0',
	X =  279.075  mm,	Y =   -438.920  mm,	Z =   -309.000  mm,
	W =  90.000 deg,	P =   0.000 deg,	R =   90.000 deg
};
P[3300]{
   GP1:
	UF : 0, UT : 6,		CONFIG : 'N U T, 0, 0, 0',
	X =  278.837  mm,	Y =   -438.900  mm,	Z =   -309.100  mm,
	W =  90.000 deg,	P =   0.000 deg,	R =   90.000 deg
};
P[3301]{
   GP1:
	UF : 0, UT : 6,		CONFIG : 'N U T, 0, 0, 0',
	X =  279.151  mm,	Y =   -439.531  mm,	Z =   -309.000  mm,
	W =  90.000 deg,	P =   0.000 deg,	R =   90.000 deg
};
P[3302]{
   GP1:
	UF : 0, UT : 6,		CONFIG : 'N U T, 0, 0, 0',
	X =  278.846  mm,	Y =   -439.516  mm,	Z =   -309.000  mm,
	W =  90.000 deg,	P =   0.000 deg,	R =   90.000 deg
};
P[3303]{
   GP1:
	UF : 0, UT : 6,		CONFIG : 'N U T, 0, 0, 0',
	X =  278.532  mm,	Y =   -439.057  mm,	Z =   -309.000  mm,
	W =  90.000 deg,	P =   0.000 deg,	R =   90.000 deg
};
P[3304]{
   GP1:
	UF : 0, UT : 6,		CONFIG : 'N U T, 0, 0, 0',
	X =  278.294  mm,	Y =   -439.184  mm,	Z =   -309.000  mm,
	W =  90.000 deg,	P =   0.000 deg,	R =   90.000 deg
};
P[3305]{
   GP1:
	UF : 0, UT : 6,		CONFIG : 'N U T, 0, 0, 0',
	X =  278.429  mm,	Y =   -439.493  mm,	Z =   -309.000  mm,
	W =  90.000 deg,	P =   0.000 deg,	R =   90.000 deg
};
P[3306]{
   GP1:
	UF : 0, UT : 6,		CONFIG : 'N U T, 0, 0, 0',
	X =  278.301  mm,	Y =   -439.381  mm,	Z =   -309.000  mm,
	W =  90.000 deg,	P =   0.000 deg,	R =   90.000 deg
};
P[3307]{
   GP1:
	UF : 0, UT : 6,		CONFIG : 'N U T, 0, 0, 0',
	X =  277.682  mm,	Y =   -439.453  mm,	Z =   -309.000  mm,
	W =  90.000 deg,	P =   0.000 deg,	R =   90.000 deg
};
P[3308]{
   GP1:
	UF : 0, UT : 6,		CONFIG : 'N U T, 0, 0, 0',
	X =  277.916  mm,	Y =   -440.035  mm,	Z =   -309.000  mm,
	W =  90.000 deg,	P =   0.000 deg,	R =   90.000 deg
};
P[3309]{
   GP1:
	UF : 0, UT : 6,		CONFIG : 'N U T, 0, 0, 0',
	X =  277.807  mm,	Y =   -439.877  mm,	Z =   -309.100  mm,
	W =  90.000 deg,	P =   0.000 deg,	R =   90.000 deg
};
P[3310]{
   GP1:
	UF : 0, UT : 6,		CONFIG : 'N U T, 0, 0, 0',
	X =  277.616  mm,	Y =   -439.807  mm,	Z =   -309.000  mm,
	W =  90.000 deg,	P =   0.000 deg,	R =   90.000 deg
};
P[3311]{
   GP1:
	UF : 0, UT : 6,		CONFIG : 'N U T, 0, 0, 0',
	X =  277.381  mm,	Y =   -440.108  mm,	Z =   -309.000  mm,
	W =  90.000 deg,	P =   0.000 deg,	R =   90.000 deg
};
P[3312]{
   GP1:
	UF : 0, UT : 6,		CONFIG : 'N U T, 0, 0, 0',
	X =  276.978  mm,	Y =   -440.524  mm,	Z =   -309.000  mm,
	W =  90.000 deg,	P =   0.000 deg,	R =   90.000 deg
};
P[3313]{
   GP1:
	UF : 0, UT : 6,		CONFIG : 'N U T, 0, 0, 0',
	X =  276.755  mm,	Y =   -440.579  mm,	Z =   -309.000  mm,
	W =  90.000 deg,	P =   0.000 deg,	R =   90.000 deg
};
P[3314]{
   GP1:
	UF : 0, UT : 6,		CONFIG : 'N U T, 0, 0, 0',
	X =  276.693  mm,	Y =   -440.522  mm,	Z =   -320.182  mm,
	W =  90.000 deg,	P =   0.000 deg,	R =   90.000 deg
};
P[3315]{
   GP1:
	UF : 0, UT : 6,		CONFIG : 'N U T, 0, 0, 0',
	X =  276.872  mm,	Y =   -440.877  mm,	Z =   -309.000  mm,
	W =  90.000 deg,	P =   0.000 deg,	R =   90.000 deg
};
P[3316]{
   GP1:
	UF : 0, UT : 6,		CONFIG : 'N U T, 0, 0, 0',
	X =  275.727  mm,	Y =   -440.491  mm,	Z =   -315.806  mm,
	W =  90.000 deg,	P =   0.000 deg,	R =   90.000 deg
};
P[3317]{
   GP1:
	UF : 0, UT : 6,		CONFIG : 'N U T, 0, 0, 0',
	X =  275.891  mm,	Y =   -441.236  mm,	Z =   -309.000  mm,
	W =  90.000 deg,	P =   0.000 deg,	R =   90.000 deg
};
P[3318]{
   GP1:
	UF : 0, UT : 6,		CONFIG : 'N U T, 0, 0, 0',
	X =  275.914  mm,	Y =   -441.357  mm,	Z =   -309.000  mm,
	W =  90.000 deg,	P =   0.000 deg,	R =   90.000 deg
};
P[3319]{
   GP1:
	UF : 0, UT : 6,		CONFIG : 'N U T, 0, 0, 0',
	X =  275.324  mm,	Y =   -441.547  mm,	Z =   -309.100  mm,
	W =  90.000 deg,	P =   0.000 deg,	R =   90.000 deg
};
P[3320]{
   GP1:
	UF : 0, UT : 6,		CONFIG : 'N U T, 0, 0, 0',
	X =  274.205  mm,	Y =   -441.939  mm,	Z =   -309.000  mm,
	W =  90.000 deg,	P =   0.000 deg,	R =   90.000 deg
};
P[3321]{
   GP1:
	UF : 0, UT : 6,		CONFIG : 'N U T, 0, 0, 0',
	X =  272.520  mm,	Y =   -442.869  mm,	Z =   -309.000  mm,
	W =  90.000 deg,	P =   0.000 deg,	R =   90.000 deg
};
P[3322]{
   GP1:
	UF : 0, UT : 6,		CONFIG : 'N U T, 0, 0, 0',
	X =  271.551  mm,	Y =   -443.443  mm,	Z =   -309.000  mm,
	W =  90.000 deg,	P =   0.000 deg,	R =   90.000 deg
};
P[3323]{
   GP1:
	UF : 0, UT : 6,		CONFIG : 'N U T, 0, 0, 0',
	X =  270.475  mm,	Y =   -443.974  mm,	Z =   -309.100  mm,
	W =  90.000 deg,	P =   0.000 deg,	R =   90.000 deg
};
P[3324]{
   GP1:
	UF : 0, UT : 6,		CONFIG : 'N U T, 0, 0, 0',
	X =  269.961  mm,	Y =   -444.835  mm,	Z =   -309.000  mm,
	W =  90.000 deg,	P =   0.000 deg,	R =   90.000 deg
};
P[3325]{
   GP1:
	UF : 0, UT : 6,		CONFIG : 'N U T, 0, 0, 0',
	X =  268.583  mm,	Y =   -445.358  mm,	Z =   -309.100  mm,
	W =  90.000 deg,	P =   0.000 deg,	R =   90.000 deg
};
P[3326]{
   GP1:
	UF : 0, UT : 6,		CONFIG : 'N U T, 0, 0, 0',
	X =  267.059  mm,	Y =   -445.797  mm,	Z =   -309.000  mm,
	W =  90.000 deg,	P =   0.000 deg,	R =   90.000 deg
};
P[3327]{
   GP1:
	UF : 0, UT : 6,		CONFIG : 'N U T, 0, 0, 0',
	X =  265.819  mm,	Y =   -446.954  mm,	Z =   -309.000  mm,
	W =  90.000 deg,	P =   0.000 deg,	R =   90.000 deg
};
P[3328]{
   GP1:
	UF : 0, UT : 6,		CONFIG : 'N U T, 0, 0, 0',
	X =  264.416  mm,	Y =   -447.597  mm,	Z =   -309.000  mm,
	W =  90.000 deg,	P =   0.000 deg,	R =   90.000 deg
};
P[3329]{
   GP1:
	UF : 0, UT : 6,		CONFIG : 'N U T, 0, 0, 0',
	X =  262.795  mm,	Y =   -448.233  mm,	Z =   -309.000  mm,
	W =  90.000 deg,	P =   0.000 deg,	R =   90.000 deg
};
P[3330]{
   GP1:
	UF : 0, UT : 6,		CONFIG : 'N U T, 0, 0, 0',
	X =  262.088  mm,	Y =   -449.181  mm,	Z =   -309.100  mm,
	W =  90.000 deg,	P =   0.000 deg,	R =   90.000 deg
};
P[3331]{
   GP1:
	UF : 0, UT : 6,		CONFIG : 'N U T, 0, 0, 0',
	X =  261.199  mm,	Y =   -449.428  mm,	Z =   -309.000  mm,
	W =  90.000 deg,	P =   0.000 deg,	R =   90.000 deg
};
P[3332]{
   GP1:
	UF : 0, UT : 6,		CONFIG : 'N U T, 0, 0, 0',
	X =  260.314  mm,	Y =   -449.954  mm,	Z =   -309.000  mm,
	W =  90.000 deg,	P =   0.000 deg,	R =   90.000 deg
};
P[3333]{
   GP1:
	UF : 0, UT : 6,		CONFIG : 'N U T, 0, 0, 0',
	X =  259.361  mm,	Y =   -450.397  mm,	Z =   -309.000  mm,
	W =  90.000 deg,	P =   0.000 deg,	R =   90.000 deg
};
P[3334]{
   GP1:
	UF : 0, UT : 6,		CONFIG : 'N U T, 0, 0, 0',
	X =  258.056  mm,	Y =   -450.663  mm,	Z =   -309.100  mm,
	W =  90.000 deg,	P =   0.000 deg,	R =   90.000 deg
};
P[3335]{
   GP1:
	UF : 0, UT : 6,		CONFIG : 'N U T, 0, 0, 0',
	X =  258.002  mm,	Y =   -451.763  mm,	Z =   -311.619  mm,
	W =  90.000 deg,	P =   0.000 deg,	R =   90.000 deg
};
P[3336]{
   GP1:
	UF : 0, UT : 6,		CONFIG : 'N U T, 0, 0, 0',
	X =  256.116  mm,	Y =   -451.844  mm,	Z =   -309.100  mm,
	W =  90.000 deg,	P =   0.000 deg,	R =   90.000 deg
};
P[3337]{
   GP1:
	UF : 0, UT : 6,		CONFIG : 'N U T, 0, 0, 0',
	X =  256.139  mm,	Y =   -452.762  mm,	Z =   -315.750  mm,
	W =  90.000 deg,	P =   0.000 deg,	R =   90.000 deg
};
P[3338]{
   GP1:
	UF : 0, UT : 6,		CONFIG : 'N U T, 0, 0, 0',
	X =  255.313  mm,	Y =   -452.862  mm,	Z =   -309.000  mm,
	W =  90.000 deg,	P =   0.000 deg,	R =   90.000 deg
};
P[3339]{
   GP1:
	UF : 0, UT : 6,		CONFIG : 'N U T, 0, 0, 0',
	X =  254.290  mm,	Y =   -453.320  mm,	Z =   -309.000  mm,
	W =  90.000 deg,	P =   0.000 deg,	R =   90.000 deg
};
P[3340]{
   GP1:
	UF : 0, UT : 6,		CONFIG : 'N U T, 0, 0, 0',
	X =  253.537  mm,	Y =   -453.731  mm,	Z =   -309.000  mm,
	W =  90.000 deg,	P =   0.000 deg,	R =   90.000 deg
};
P[3341]{
   GP1:
	UF : 0, UT : 6,		CONFIG : 'N U T, 0, 0, 0',
	X =  252.115  mm,	Y =   -454.208  mm,	Z =   -309.000  mm,
	W =  90.000 deg,	P =   0.000 deg,	R =   90.000 deg
};
P[3342]{
   GP1:
	UF : 0, UT : 6,		CONFIG : 'N U T, 0, 0, 0',
	X =  251.265  mm,	Y =   -455.339  mm,	Z =   -309.000  mm,
	W =  90.000 deg,	P =   0.000 deg,	R =   90.000 deg
};
P[3343]{
   GP1:
	UF : 0, UT : 6,		CONFIG : 'N U T, 0, 0, 0',
	X =  250.427  mm,	Y =   -456.091  mm,	Z =   -309.404  mm,
	W =  90.000 deg,	P =   0.000 deg,	R =   90.000 deg
};
P[3344]{
   GP1:
	UF : 0, UT : 6,		CONFIG : 'N U T, 0, 0, 0',
	X =  249.062  mm,	Y =   -456.723  mm,	Z =   -309.100  mm,
	W =  90.000 deg,	P =   0.000 deg,	R =   90.000 deg
};
P[3345]{
   GP1:
	UF : 0, UT : 6,		CONFIG : 'N U T, 0, 0, 0',
	X =  247.885  mm,	Y =   -456.753  mm,	Z =   -309.000  mm,
	W =  90.000 deg,	P =   0.000 deg,	R =   90.000 deg
};
P[3346]{
   GP1:
	UF : 0, UT : 6,		CONFIG : 'N U T, 0, 0, 0',
	X =  247.270  mm,	Y =   -457.497  mm,	Z =   -309.000  mm,
	W =  90.000 deg,	P =   0.000 deg,	R =   90.000 deg
};
P[3347]{
   GP1:
	UF : 0, UT : 6,		CONFIG : 'N U T, 0, 0, 0',
	X =  246.542  mm,	Y =   -457.699  mm,	Z =   -317.201  mm,
	W =  90.000 deg,	P =   0.000 deg,	R =   90.000 deg
};
P[3348]{
   GP1:
	UF : 0, UT : 6,		CONFIG : 'N U T, 0, 0, 0',
	X =  245.101  mm,	Y =   -458.390  mm,	Z =   -309.000  mm,
	W =  90.000 deg,	P =   0.000 deg,	R =   90.000 deg
};
P[3349]{
   GP1:
	UF : 0, UT : 6,		CONFIG : 'N U T, 0, 0, 0',
	X =  244.155  mm,	Y =   -459.061  mm,	Z =   -309.000  mm,
	W =  90.000 deg,	P =   0.000 deg,	R =   90.000 deg
};
P[3350]{
   GP1:
	UF : 0, UT : 6,		CONFIG : 'N U T, 0, 0, 0',
	X =  242.157  mm,	Y =   -460.162  mm,	Z =   -309.100  mm,
	W =  90.000 deg,	P =   0.000 deg,	R =   90.000 deg
};
P[3351]{
   GP1:
	UF : 0, UT : 6,		CONFIG : 'N U T, 0, 0, 0',
	X =  241.362  mm,	Y =   -460.588  mm,	Z =   -309.000  mm,
	W =  90.000 deg,	P =   0.000 deg,	R =   90.000 deg
};
P[3352]{
   GP1:
	UF : 0, UT : 6,		CONFIG : 'N U T, 0, 0, 0',
	X =  240.253  mm,	Y =   -461.771  mm,	Z =   -309.100  mm,
	W =  90.000 deg,	P =   0.000 deg,	R =   90.000 deg
};
P[3353]{
   GP1:
	UF : 0, UT : 6,		CONFIG : 'N U T, 0, 0, 0',
	X =  238.984  mm,	Y =   -462.133  mm,	Z =   -309.100  mm,
	W =  90.000 deg,	P =   0.000 deg,	R =   90.000 deg
};
P[3354]{
   GP1:
	UF : 0, UT : 6,		CONFIG : 'N U T, 0, 0, 0',
	X =  238.398  mm,	Y =   -462.993  mm,	Z =   -309.000  mm,
	W =  90.000 deg,	P =   0.000 deg,	R =   90.000 deg
};
P[3355]{
   GP1:
	UF : 0, UT : 6,		CONFIG : 'N U T, 0, 0, 0',
	X =  237.655  mm,	Y =   -462.918  mm,	Z =   -309.000  mm,
	W =  90.000 deg,	P =   0.000 deg,	R =   90.000 deg
};
P[3356]{
   GP1:
	UF : 0, UT : 6,		CONFIG : 'N U T, 0, 0, 0',
	X =  237.080  mm,	Y =   -463.517  mm,	Z =   -309.000  mm,
	W =  90.000 deg,	P =   0.000 deg,	R =   90.000 deg
};
P[3357]{
   GP1:
	UF : 0, UT : 6,		CONFIG : 'N U T, 0, 0, 0',
	X =  235.960  mm,	Y =   -463.844  mm,	Z =   -309.000  mm,
	W =  90.000 deg,	P =   0.000 deg,	R =   90.000 deg
};
P[3358]{
   GP1:
	UF : 0, UT : 6,		CONFIG : 'N U T, 0, 0, 0',
	X =  235.094  mm,	Y =   -464.401  mm,	Z =   -309.000  mm,
	W =  90.000 deg,	P =   0.000 deg,	R =   90.000 deg
};
P[3359]{
   GP1:
	UF : 0, UT : 6,		CONFIG : 'N U T, 0, 0, 0',
	X =  234.195  mm,	Y =   -464.983  mm,	Z =   -309.000  mm,
	W =  90.000 deg,	P =   0.000 deg,	R =   90.000 deg
};
P[3360]{
   GP1:
	UF : 0, UT : 6,		CONFIG : 'N U T, 0, 0, 0',
	X =  233.258  mm,	Y =   -465.698  mm,	Z =   -311.006  mm,
	W =  90.000 deg,	P =   0.000 deg,	R =   90.000 deg
};
P[3361]{
   GP1:
	UF : 0, UT : 6,		CONFIG : 'N U T, 0, 0, 0',
	X =  232.349  mm,	Y =   -465.948  mm,	Z =   -309.000  mm,
	W =  90.000 deg,	P =   0.000 deg,	R =   90.000 deg
};
P[3362]{
   GP1:
	UF : 0, UT : 6,		CONFIG : 'N U T, 0, 0, 0',
	X =  231.479  mm,	Y =   -466.435  mm,	Z =   -309.000  mm,
	W =  90.000 deg,	P =   0.000 deg,	R =   90.000 deg
};
P[3363]{
   GP1:
	UF : 0, UT : 6,		CONFIG : 'N U T, 0, 0, 0',
	X =  230.705  mm,	Y =   -466.900  mm,	Z =   -309.000  mm,
	W =  90.000 deg,	P =   0.000 deg,	R =   90.000 deg
};
P[3364]{
   GP1:
	UF : 0, UT : 6,		CONFIG : 'N U T, 0, 0, 0',
	X =  229.847  mm,	Y =   -467.161  mm,	Z =   -309.000  mm,
	W =  90.000 deg,	P =   0.000 deg,	R =   90.000 deg
};
P[3365]{
   GP1:
	UF : 0, UT : 6,		CONFIG : 'N U T, 0, 0, 0',
	X =  229.828  mm,	Y =   -467.563  mm,	Z =   -309.000  mm,
	W =  90.000 deg,	P =   0.000 deg,	R =   90.000 deg
};
P[3366]{
   GP1:
	UF : 0, UT : 6,		CONFIG : 'N U T, 0, 0, 0',
	X =  229.866  mm,	Y =   -467.709  mm,	Z =   -309.100  mm,
	W =  90.000 deg,	P =   0.000 deg,	R =   90.000 deg
};
P[3367]{
   GP1:
	UF : 0, UT : 6,		CONFIG : 'N U T, 0, 0, 0',
	X =  229.891  mm,	Y =   -467.912  mm,	Z =   -309.000  mm,
	W =  90.000 deg,	P =   0.000 deg,	R =   90.000 deg
};
P[3368]{
   GP1:
	UF : 0, UT : 6,		CONFIG : 'N U T, 0, 0, 0',
	X =  229.464  mm,	Y =   -467.631  mm,	Z =   -309.000  mm,
	W =  90.000 deg,	P =   0.000 deg,	R =   90.000 deg
};
P[3369]{
   GP1:
	UF : 0, UT : 6,		CONFIG : 'N U T, 0, 0, 0',
	X =  229.046  mm,	Y =   -467.373  mm,	Z =   -309.000  mm,
	W =  90.000 deg,	P =   0.000 deg,	R =   90.000 deg
};
P[3370]{
   GP1:
	UF : 0, UT : 6,		CONFIG : 'N U T, 0, 0, 0',
	X =  229.336  mm,	Y =   -468.249  mm,	Z =   -311.188  mm,
	W =  90.000 deg,	P =   0.000 deg,	R =   90.000 deg
};
P[3371]{
   GP1:
	UF : 0, UT : 6,		CONFIG : 'N U T, 0, 0, 0',
	X =  228.968  mm,	Y =   -467.803  mm,	Z =   -309.100  mm,
	W =  90.000 deg,	P =   0.000 deg,	R =   90.000 deg
};
P[3372]{
   GP1:
	UF : 0, UT : 6,		CONFIG : 'N U T, 0, 0, 0',
	X =  228.688  mm,	Y =   -467.707  mm,	Z =   -309.100  mm,
	W =  90.000 deg,	P =   0.000 deg,	R =   90.000 deg
};
P[3373]{
   GP1:
	UF : 0, UT : 6,		CONFIG : 'N U T, 0, 0, 0',
	X =  228.740  mm,	Y =   -468.070  mm,	Z =   -309.000  mm,
	W =  90.000 deg,	P =   0.000 deg,	R =   90.000 deg
};
P[3374]{
   GP1:
	UF : 0, UT : 6,		CONFIG : 'N U T, 0, 0, 0',
	X =  228.269  mm,	Y =   -468.472  mm,	Z =   -309.000  mm,
	W =  90.000 deg,	P =   0.000 deg,	R =   90.000 deg
};
P[3375]{
   GP1:
	UF : 0, UT : 6,		CONFIG : 'N U T, 0, 0, 0',
	X =  227.905  mm,	Y =   -468.156  mm,	Z =   -309.000  mm,
	W =  90.000 deg,	P =   0.000 deg,	R =   90.000 deg
};
P[3376]{
   GP1:
	UF : 0, UT : 6,		CONFIG : 'N U T, 0, 0, 0',
	X =  227.920  mm,	Y =   -468.786  mm,	Z =   -309.100  mm,
	W =  90.000 deg,	P =   0.000 deg,	R =   90.000 deg
};
P[3377]{
   GP1:
	UF : 0, UT : 6,		CONFIG : 'N U T, 0, 0, 0',
	X =  227.481  mm,	Y =   -468.382  mm,	Z =   -309.000  mm,
	W =  90.000 deg,	P =   0.000 deg,	R =   90.000 deg
};
P[3378]{
   GP1:
	UF : 0, UT : 6,		CONFIG : 'N U T, 0, 0, 0',
	X =  227.695  mm,	Y =   -469.197  mm,	Z =   -309.100  mm,
	W =  90.000 deg,	P =   0.000 deg,	R =   90.000 deg
};
P[3379]{
   GP1:
	UF : 0, UT : 6,		CONFIG : 'N U T, 0, 0, 0',
	X =  226.881  mm,	Y =   -468.653  mm,	Z =   -309.344  mm,
	W =  90.000 deg,	P =   0.000 deg,	R =   90.000 deg
};
P[3380]{
   GP1:
	UF : 0, UT : 6,		CONFIG : 'N U T, 0, 0, 0',
	X =  226.945  mm,	Y =   -468.938  mm,	Z =   -309.000  mm,
	W =  90.000 deg,	P =   0.000 deg,	R =   90.000 deg
};
P[3381]{
   GP1:
	UF : 0, UT : 6,		CONFIG : 'N U T, 0, 0, 0',
	X =  226.507  mm,	Y =   -469.334  mm,	Z =   -309.000  mm,
	W =  90.000 deg,	P =   0.000 deg,	R =   90.000 deg
};
P[3382]{
   GP1:
	UF : 0, UT : 6,		CONFIG : 'N U T, 0, 0, 0',
	X =  225.921  mm,	Y =   -470.015  mm,	Z =   -309.000  mm,
	W =  90.000 deg,	P =   0.000 deg,	R =   90.000 deg
};
P[3383]{
   GP1:
	UF : 0, UT : 6,		CONFIG : 'N U T, 0, 0, 0',
	X =  225.207  mm,	Y =   -469.571  mm,	Z =   -309.000  mm,
	W =  90.000 deg,	P =   0.000 deg,	R =   90.000 deg
};
P[3384]{
   GP1:
	UF : 0, UT : 6,		CONFIG : 'N U T, 0, 0, 0',
	X =  224.979  mm,	Y =   -470.636  mm,	Z =   -309.100  mm,
	W =  90.000 deg,	P =   0.000 deg,	R =   90.000 deg
};
P[3385]{
   GP1:
	UF : 0, UT : 6,		CONFIG : 'N U T, 0, 0, 0',
	X =  224.574  mm,	Y =   -470.261  mm,	Z =   -324.425  mm,
	W =  90.000 deg,	P =   0.000 deg,	R =   90.000 deg
};
P[3386]{
   GP1:
	UF : 0, UT : 6,		CONFIG : 'N U T, 0, 0, 0',
	X =  224.050  mm,	Y =   -471.070  mm,	Z =   -309.100  mm,
	W =  90.000 deg,	P =   0.000 deg,	R =   90.000 deg
};
P[3387]{
   GP1:
	UF : 0, UT : 6,		CONFIG : 'N U T, 0, 0, 0',
	X =  223.375  mm,	Y =   -471.399  mm,	Z =   -309.000  mm,
	W =  90.000 deg,	P =   0.000 deg,	R =   90.000 deg
};
P[3388]{
   GP1:
	UF : 0, UT : 6,		CONFIG : 'N U T, 0, 0, 0',
	X =  222.698  mm,	Y =   -471.310  mm,	Z =   -326.914  mm,
	W =  90.000 deg,	P =   0.000 deg,	R =   90.000 deg
};
P[3389]{
   GP1:
	UF : 0, UT : 6,		CONFIG : 'N U T, 0, 0, 0',
	X =  222.206  mm,	Y =   -471.714  mm,	Z =   -309.000  mm,
	W =  90.000 deg,	P =   0.000 deg,	R =   90.000 deg
};
P[3390]{
   GP1:
	UF : 0, UT : 6,		CONFIG : 'N U T, 0, 0, 0',
	X =  221.113  mm,	Y =   -472.371  mm,	Z =   -309.000  mm,
	W =  90.000 deg,	P =   0.000 deg,	R =   90.000 deg
};
P[3391]{
   GP1:
	UF : 0, UT : 6,		CONFIG : 'N U T, 0, 0, 0',
	X =  220.317  mm,	Y =   -472.805  mm,	Z =   -309.000  mm,
	W =  90.000 deg,	P =   0.000 deg,	R =   90.000 deg
};
P[3392]{
   GP1:
	UF : 0, UT : 6,		CONFIG : 'N U T, 0, 0, 0',
	X =  220.568  mm,	Y =   -473.280  mm,	Z =   -309.000  mm,
	W =  90.000 deg,	P =   0.000 deg,	R =   90.000 deg
};
P[3393]{
   GP1:
	UF : 0, UT : 6,		CONFIG : 'N U T, 0, 0, 0',
	X =  219.376  mm,	Y =   -473.461  mm,	Z =   -309.000  mm,
	W =  90.000 deg,	P =   0.000 deg,	R =   90.000 deg
};
P[3394]{
   GP1:
	UF : 0, UT : 6,		CONFIG : 'N U T, 0, 0, 0',
	X =  218.936  mm,	Y =   -474.026  mm,	Z =   -309.100  mm,
	W =  90.000 deg,	P =   0.000 deg,	R =   90.000 deg
};
P[3395]{
   GP1:
	UF : 0, UT : 6,		CONFIG : 'N U T, 0, 0, 0',
	X =  217.962  mm,	Y =   -474.156  mm,	Z =   -309.000  mm,
	W =  90.000 deg,	P =   0.000 deg,	R =   90.000 deg
};
P[3396]{
   GP1:
	UF : 0, UT : 6,		CONFIG : 'N U T, 0, 0, 0',
	X =  217.767  mm,	Y =   -474.880  mm,	Z =   -309.100  mm,
	W =  90.000 deg,	P =   0.000 deg,	R =   90.000 deg
};
P[3397]{
   GP1:
	UF : 0, UT : 6,		CONFIG : 'N U T, 0, 0, 0',
	X =  217.097  mm,	Y =   -474.449  mm,	Z =   -309.000  mm,
	W =  90.000 deg,	P =   0.000 deg,	R =   90.000 deg
};
P[3398]{
   GP1:
	UF : 0, UT : 6,		CONFIG : 'N U T, 0, 0, 0',
	X =  217.033  mm,	Y =   -474.992  mm,	Z =   -309.100  mm,
	W =  90.000 deg,	P =   0.000 deg,	R =   90.000 deg
};
P[3399]{
   GP1:
	UF : 0, UT : 6,		CONFIG : 'N U T, 0, 0, 0',
	X =  216.279  mm,	Y =   -475.594  mm,	Z =   -309.100  mm,
	W =  90.000 deg,	P =   0.000 deg,	R =   90.000 deg
};
P[3400]{
   GP1:
	UF : 0, UT : 6,		CONFIG : 'N U T, 0, 0, 0',
	X =  215.282  mm,	Y =   -475.703  mm,	Z =   -309.000  mm,
	W =  90.000 deg,	P =   0.000 deg,	R =   90.000 deg
};
P[3401]{
   GP1:
	UF : 0, UT : 6,		CONFIG : 'N U T, 0, 0, 0',
	X =  215.078  mm,	Y =   -476.238  mm,	Z =   -324.184  mm,
	W =  90.000 deg,	P =   0.000 deg,	R =   90.000 deg
};
P[3402]{
   GP1:
	UF : 0, UT : 6,		CONFIG : 'N U T, 0, 0, 0',
	X =  214.064  mm,	Y =   -476.584  mm,	Z =   -309.000  mm,
	W =  90.000 deg,	P =   0.000 deg,	R =   90.000 deg
};
P[3403]{
   GP1:
	UF : 0, UT : 6,		CONFIG : 'N U T, 0, 0, 0',
	X =  213.427  mm,	Y =   -476.835  mm,	Z =   -309.000  mm,
	W =  90.000 deg,	P =   0.000 deg,	R =   90.000 deg
};
P[3404]{
   GP1:
	UF : 0, UT : 6,		CONFIG : 'N U T, 0, 0, 0',
	X =  212.551  mm,	Y =   -477.641  mm,	Z =   -309.000  mm,
	W =  90.000 deg,	P =   0.000 deg,	R =   90.000 deg
};
P[3405]{
   GP1:
	UF : 0, UT : 6,		CONFIG : 'N U T, 0, 0, 0',
	X =  211.558  mm,	Y =   -477.493  mm,	Z =   -309.000  mm,
	W =  90.000 deg,	P =   0.000 deg,	R =   90.000 deg
};
P[3406]{
   GP1:
	UF : 0, UT : 6,		CONFIG : 'N U T, 0, 0, 0',
	X =  211.839  mm,	Y =   -478.089  mm,	Z =   -309.050  mm,
	W =  90.000 deg,	P =   0.000 deg,	R =   90.000 deg
};
P[3407]{
   GP1:
	UF : 0, UT : 6,		CONFIG : 'N U T, 0, 0, 0',
	X =  210.946  mm,	Y =   -478.556  mm,	Z =   -327.700  mm,
	W =  90.000 deg,	P =   0.000 deg,	R =   90.000 deg
};
P[3408]{
   GP1:
	UF : 0, UT : 6,		CONFIG : 'N U T, 0, 0, 0',
	X =  210.651  mm,	Y =   -478.191  mm,	Z =   -309.000  mm,
	W =  90.000 deg,	P =   0.000 deg,	R =   90.000 deg
};
P[3409]{
   GP1:
	UF : 0, UT : 6,		CONFIG : 'N U T, 0, 0, 0',
	X =  209.531  mm,	Y =   -478.989  mm,	Z =   -309.100  mm,
	W =  90.000 deg,	P =   0.000 deg,	R =   90.000 deg
};
P[3410]{
   GP1:
	UF : 0, UT : 6,		CONFIG : 'N U T, 0, 0, 0',
	X =  209.103  mm,	Y =   -478.884  mm,	Z =   -309.000  mm,
	W =  90.000 deg,	P =   0.000 deg,	R =   90.000 deg
};
P[3411]{
   GP1:
	UF : 0, UT : 6,		CONFIG : 'N U T, 0, 0, 0',
	X =  209.222  mm,	Y =   -479.603  mm,	Z =   -309.100  mm,
	W =  90.000 deg,	P =   0.000 deg,	R =   90.000 deg
};
P[3412]{
   GP1:
	UF : 0, UT : 6,		CONFIG : 'N U T, 0, 0, 0',
	X =  208.375  mm,	Y =   -479.782  mm,	Z =   -309.000  mm,
	W =  90.000 deg,	P =   0.000 deg,	R =   90.000 deg
};
P[3413]{
   GP1:
	UF : 0, UT : 6,		CONFIG : 'N U T, 0, 0, 0',
	X =  207.346  mm,	Y =   -480.439  mm,	Z =   -309.000  mm,
	W =  90.000 deg,	P =   0.000 deg,	R =   90.000 deg
};
P[3414]{
   GP1:
	UF : 0, UT : 6,		CONFIG : 'N U T, 0, 0, 0',
	X =  206.217  mm,	Y =   -480.866  mm,	Z =   -309.000  mm,
	W =  90.000 deg,	P =   0.000 deg,	R =   90.000 deg
};
P[3415]{
   GP1:
	UF : 0, UT : 6,		CONFIG : 'N U T, 0, 0, 0',
	X =  205.980  mm,	Y =   -481.549  mm,	Z =   -312.901  mm,
	W =  90.000 deg,	P =   0.000 deg,	R =   90.000 deg
};
P[3416]{
   GP1:
	UF : 0, UT : 6,		CONFIG : 'N U T, 0, 0, 0',
	X =  205.518  mm,	Y =   -481.319  mm,	Z =   -309.050  mm,
	W =  90.000 deg,	P =   0.000 deg,	R =   90.000 deg
};
P[3417]{
   GP1:
	UF : 0, UT : 6,		CONFIG : 'N U T, 0, 0, 0',
	X =  204.866  mm,	Y =   -481.684  mm,	Z =   -309.100  mm,
	W =  90.000 deg,	P =   0.000 deg,	R =   90.000 deg
};
P[3418]{
   GP1:
	UF : 0, UT : 6,		CONFIG : 'N U T, 0, 0, 0',
	X =  204.972  mm,	Y =   -482.156  mm,	Z =   -327.903  mm,
	W =  90.000 deg,	P =   0.000 deg,	R =   90.000 deg
};
P[3419]{
   GP1:
	UF : 0, UT : 6,		CONFIG : 'N U T, 0, 0, 0',
	X =  204.185  mm,	Y =   -481.972  mm,	Z =   -309.000  mm,
	W =  90.000 deg,	P =   0.000 deg,	R =   90.000 deg
};
P[3420]{
   GP1:
	UF : 0, UT : 6,		CONFIG : 'N U T, 0, 0, 0',
	X =  204.266  mm,	Y =   -482.560  mm,	Z =   -309.100  mm,
	W =  90.000 deg,	P =   0.000 deg,	R =   90.000 deg
};
P[3421]{
   GP1:
	UF : 0, UT : 6,		CONFIG : 'N U T, 0, 0, 0',
	X =  203.470  mm,	Y =   -482.734  mm,	Z =   -309.000  mm,
	W =  90.000 deg,	P =   0.000 deg,	R =   90.000 deg
};
P[3422]{
   GP1:
	UF : 0, UT : 6,		CONFIG : 'N U T, 0, 0, 0',
	X =  202.751  mm,	Y =   -482.593  mm,	Z =   -309.000  mm,
	W =  90.000 deg,	P =   0.000 deg,	R =   90.000 deg
};
P[3423]{
   GP1:
	UF : 0, UT : 6,		CONFIG : 'N U T, 0, 0, 0',
	X =  202.732  mm,	Y =   -483.103  mm,	Z =   -309.000  mm,
	W =  90.000 deg,	P =   0.000 deg,	R =   90.000 deg
};
P[3424]{
   GP1:
	UF : 0, UT : 6,		CONFIG : 'N U T, 0, 0, 0',
	X =  202.361  mm,	Y =   -483.672  mm,	Z =   -309.100  mm,
	W =  90.000 deg,	P =   0.000 deg,	R =   90.000 deg
};
P[3425]{
   GP1:
	UF : 0, UT : 6,		CONFIG : 'N U T, 0, 0, 0',
	X =  201.883  mm,	Y =   -483.416  mm,	Z =   -309.000  mm,
	W =  90.000 deg,	P =   0.000 deg,	R =   90.000 deg
};
P[3426]{
   GP1:
	UF : 0, UT : 6,		CONFIG : 'N U T, 0, 0, 0',
	X =  201.503  mm,	Y =   -484.280  mm,	Z =   -309.000  mm,
	W =  90.000 deg,	P =   0.000 deg,	R =   90.000 deg
};
P[3427]{
   GP1:
	UF : 0, UT : 6,		CONFIG : 'N U T, 0, 0, 0',
	X =  200.979  mm,	Y =   -484.024  mm,	Z =   -309.000  mm,
	W =  90.000 deg,	P =   0.000 deg,	R =   90.000 deg
};
P[3428]{
   GP1:
	UF : 0, UT : 6,		CONFIG : 'N U T, 0, 0, 0',
	X =  200.855  mm,	Y =   -484.697  mm,	Z =   -309.000  mm,
	W =  90.000 deg,	P =   0.000 deg,	R =   90.000 deg
};
P[3429]{
   GP1:
	UF : 0, UT : 6,		CONFIG : 'N U T, 0, 0, 0',
	X =  200.318  mm,	Y =   -484.205  mm,	Z =   -312.782  mm,
	W =  90.000 deg,	P =   0.000 deg,	R =   90.000 deg
};
P[3430]{
   GP1:
	UF : 0, UT : 6,		CONFIG : 'N U T, 0, 0, 0',
	X =  200.026  mm,	Y =   -484.142  mm,	Z =   -309.100  mm,
	W =  90.000 deg,	P =   0.000 deg,	R =   90.000 deg
};
P[3431]{
   GP1:
	UF : 0, UT : 6,		CONFIG : 'N U T, 0, 0, 0',
	X =  199.866  mm,	Y =   -484.968  mm,	Z =   -309.100  mm,
	W =  90.000 deg,	P =   0.000 deg,	R =   90.000 deg
};
P[3432]{
   GP1:
	UF : 0, UT : 6,		CONFIG : 'N U T, 0, 0, 0',
	X =  199.499  mm,	Y =   -484.683  mm,	Z =   -309.100  mm,
	W =  90.000 deg,	P =   0.000 deg,	R =   90.000 deg
};
P[3433]{
   GP1:
	UF : 0, UT : 6,		CONFIG : 'N U T, 0, 0, 0',
	X =  199.010  mm,	Y =   -484.781  mm,	Z =   -309.000  mm,
	W =  90.000 deg,	P =   0.000 deg,	R =   90.000 deg
};
P[3434]{
   GP1:
	UF : 0, UT : 6,		CONFIG : 'N U T, 0, 0, 0',
	X =  199.128  mm,	Y =   -485.590  mm,	Z =   -309.000  mm,
	W =  90.000 deg,	P =   0.000 deg,	R =   90.000 deg
};
P[3435]{
   GP1:
	UF : 0, UT : 6,		CONFIG : 'N U T, 0, 0, 0',
	X =  198.800  mm,	Y =   -485.362  mm,	Z =   -309.000  mm,
	W =  90.000 deg,	P =   0.000 deg,	R =   90.000 deg
};
P[3436]{
   GP1:
	UF : 0, UT : 6,		CONFIG : 'N U T, 0, 0, 0',
	X =  197.969  mm,	Y =   -485.700  mm,	Z =   -309.000  mm,
	W =  90.000 deg,	P =   0.000 deg,	R =   90.000 deg
};
P[3437]{
   GP1:
	UF : 0, UT : 6,		CONFIG : 'N U T, 0, 0, 0',
	X =  197.584  mm,	Y =   -485.549  mm,	Z =   -309.000  mm,
	W =  90.000 deg,	P =   0.000 deg,	R =   90.000 deg
};
P[3438]{
   GP1:
	UF : 0, UT : 6,		CONFIG : 'N U T, 0, 0, 0',
	X =  197.497  mm,	Y =   -485.805  mm,	Z =   -309.100  mm,
	W =  90.000 deg,	P =   0.000 deg,	R =   90.000 deg
};
P[3439]{
   GP1:
	UF : 0, UT : 6,		CONFIG : 'N U T, 0, 0, 0',
	X =  197.671  mm,	Y =   -486.384  mm,	Z =   -309.100  mm,
	W =  90.000 deg,	P =   0.000 deg,	R =   90.000 deg
};
P[3440]{
   GP1:
	UF : 0, UT : 6,		CONFIG : 'N U T, 0, 0, 0',
	X =  196.988  mm,	Y =   -486.325  mm,	Z =   -309.000  mm,
	W =  90.000 deg,	P =   0.000 deg,	R =   90.000 deg
};
P[3441]{
   GP1:
	UF : 0, UT : 6,		CONFIG : 'N U T, 0, 0, 0',
	X =  196.797  mm,	Y =   -486.118  mm,	Z =   -309.000  mm,
	W =  90.000 deg,	P =   0.000 deg,	R =   90.000 deg
};
P[3442]{
   GP1:
	UF : 0, UT : 6,		CONFIG : 'N U T, 0, 0, 0',
	X =  196.729  mm,	Y =   -486.332  mm,	Z =   -309.100  mm,
	W =  90.000 deg,	P =   0.000 deg,	R =   90.000 deg
};
P[3443]{
   GP1:
	UF : 0, UT : 6,		CONFIG : 'N U T, 0, 0, 0',
	X =  196.980  mm,	Y =   -486.900  mm,	Z =   -309.100  mm,
	W =  90.000 deg,	P =   0.000 deg,	R =   90.000 deg
};
P[3444]{
   GP1:
	UF : 0, UT : 6,		CONFIG : 'N U T, 0, 0, 0',
	X =  196.703  mm,	Y =   -486.855  mm,	Z =   -309.000  mm,
	W =  90.000 deg,	P =   0.000 deg,	R =   90.000 deg
};
P[3445]{
   GP1:
	UF : 0, UT : 6,		CONFIG : 'N U T, 0, 0, 0',
	X =  196.299  mm,	Y =   -486.934  mm,	Z =   -309.000  mm,
	W =  90.000 deg,	P =   0.000 deg,	R =   90.000 deg
};
P[3446]{
   GP1:
	UF : 0, UT : 6,		CONFIG : 'N U T, 0, 0, 0',
	X =  195.967  mm,	Y =   -486.560  mm,	Z =   -309.000  mm,
	W =  90.000 deg,	P =   0.000 deg,	R =   90.000 deg
};
P[3447]{
   GP1:
	UF : 0, UT : 6,		CONFIG : 'N U T, 0, 0, 0',
	X =  196.084  mm,	Y =   -486.830  mm,	Z =   -309.000  mm,
	W =  90.000 deg,	P =   0.000 deg,	R =   90.000 deg
};
P[3448]{
   GP1:
	UF : 0, UT : 6,		CONFIG : 'N U T, 0, 0, 0',
	X =  195.925  mm,	Y =   -486.810  mm,	Z =   -309.000  mm,
	W =  90.000 deg,	P =   0.000 deg,	R =   90.000 deg
};
P[3449]{
   GP1:
	UF : 0, UT : 6,		CONFIG : 'N U T, 0, 0, 0',
	X =  195.717  mm,	Y =   -487.612  mm,	Z =   -309.000  mm,
	W =  90.000 deg,	P =   0.000 deg,	R =   90.000 deg
};
P[3450]{
   GP1:
	UF : 0, UT : 6,		CONFIG : 'N U T, 0, 0, 0',
	X =  195.396  mm,	Y =   -487.271  mm,	Z =   -309.000  mm,
	W =  90.000 deg,	P =   0.000 deg,	R =   90.000 deg
};
P[3451]{
   GP1:
	UF : 0, UT : 6,		CONFIG : 'N U T, 0, 0, 0',
	X =  195.484  mm,	Y =   -487.551  mm,	Z =   -309.100  mm,
	W =  90.000 deg,	P =   0.000 deg,	R =   90.000 deg
};
P[3452]{
   GP1:
	UF : 0, UT : 6,		CONFIG : 'N U T, 0, 0, 0',
	X =  195.288  mm,	Y =   -487.488  mm,	Z =   -309.000  mm,
	W =  90.000 deg,	P =   0.000 deg,	R =   90.000 deg
};
P[3453]{
   GP1:
	UF : 0, UT : 6,		CONFIG : 'N U T, 0, 0, 0',
	X =  194.963  mm,	Y =   -487.536  mm,	Z =   -309.000  mm,
	W =  90.000 deg,	P =   0.000 deg,	R =   90.000 deg
};
P[3454]{
   GP1:
	UF : 0, UT : 6,		CONFIG : 'N U T, 0, 0, 0',
	X =  194.991  mm,	Y =   -488.058  mm,	Z =   -309.000  mm,
	W =  90.000 deg,	P =   0.000 deg,	R =   90.000 deg
};
P[3455]{
   GP1:
	UF : 0, UT : 6,		CONFIG : 'N U T, 0, 0, 0',
	X =  194.583  mm,	Y =   -488.094  mm,	Z =   -309.000  mm,
	W =  90.000 deg,	P =   0.000 deg,	R =   90.000 deg
};
P[3456]{
   GP1:
	UF : 0, UT : 6,		CONFIG : 'N U T, 0, 0, 0',
	X =  194.264  mm,	Y =   -487.785  mm,	Z =   -309.100  mm,
	W =  90.000 deg,	P =   0.000 deg,	R =   90.000 deg
};
P[3457]{
   GP1:
	UF : 0, UT : 6,		CONFIG : 'N U T, 0, 0, 0',
	X =  194.394  mm,	Y =   -488.104  mm,	Z =   -309.000  mm,
	W =  90.000 deg,	P =   0.000 deg,	R =   90.000 deg
};
P[3458]{
   GP1:
	UF : 0, UT : 6,		CONFIG : 'N U T, 0, 0, 0',
	X =  193.778  mm,	Y =   -488.342  mm,	Z =   -309.000  mm,
	W =  90.000 deg,	P =   0.000 deg,	R =   90.000 deg
};
P[3459]{
   GP1:
	UF : 0, UT : 6,		CONFIG : 'N U T, 0, 0, 0',
	X =  193.852  mm,	Y =   -488.697  mm,	Z =   -309.000  mm,
	W =  90.000 deg,	P =   0.000 deg,	R =   90.000 deg
};
P[3460]{
   GP1:
	UF : 0, UT : 6,		CONFIG : 'N U T, 0, 0, 0',
	X =  193.402  mm,	Y =   -488.920  mm,	Z =   -309.100  mm,
	W =  90.000 deg,	P =   0.000 deg,	R =   90.000 deg
};
P[3461]{
   GP1:
	UF : 0, UT : 6,		CONFIG : 'N U T, 0, 0, 0',
	X =  192.917  mm,	Y =   -488.676  mm,	Z =   -325.074  mm,
	W =  90.000 deg,	P =   0.000 deg,	R =   90.000 deg
};
P[3462]{
   GP1:
	UF : 0, UT : 6,		CONFIG : 'N U T, 0, 0, 0',
	X =  192.752  mm,	Y =   -489.451  mm,	Z =   -309.000  mm,
	W =  90.000 deg,	P =   0.000 deg,	R =   90.000 deg
};
P[3463]{
   GP1:
	UF : 0, UT : 6,		CONFIG : 'N U T, 0, 0, 0',
	X =  191.890  mm,	Y =   -489.408  mm,	Z =   -309.000  mm,
	W =  90.000 deg,	P =   0.000 deg,	R =   90.000 deg
};
P[3464]{
   GP1:
	UF : 0, UT : 6,		CONFIG : 'N U T, 0, 0, 0',
	X =  190.851  mm,	Y =   -489.933  mm,	Z =   -309.100  mm,
	W =  90.000 deg,	P =   0.000 deg,	R =   90.000 deg
};
P[3465]{
   GP1:
	UF : 0, UT : 6,		CONFIG : 'N U T, 0, 0, 0',
	X =  189.731  mm,	Y =   -490.970  mm,	Z =   -323.887  mm,
	W =  90.000 deg,	P =   0.000 deg,	R =   90.000 deg
};
P[3466]{
   GP1:
	UF : 0, UT : 6,		CONFIG : 'N U T, 0, 0, 0',
	X =  188.830  mm,	Y =   -491.364  mm,	Z =   -312.801  mm,
	W =  90.000 deg,	P =   0.000 deg,	R =   90.000 deg
};
P[3467]{
   GP1:
	UF : 0, UT : 6,		CONFIG : 'N U T, 0, 0, 0',
	X =  188.000  mm,	Y =   -491.052  mm,	Z =   -309.000  mm,
	W =  90.000 deg,	P =   0.000 deg,	R =   90.000 deg
};
P[3468]{
   GP1:
	UF : 0, UT : 6,		CONFIG : 'N U T, 0, 0, 0',
	X =  187.486  mm,	Y =   -491.974  mm,	Z =   -309.000  mm,
	W =  90.000 deg,	P =   0.000 deg,	R =   90.000 deg
};
P[3469]{
   GP1:
	UF : 0, UT : 6,		CONFIG : 'N U T, 0, 0, 0',
	X =  185.118  mm,	Y =   -493.278  mm,	Z =   -309.000  mm,
	W =  90.000 deg,	P =   0.000 deg,	R =   90.000 deg
};
P[3470]{
   GP1:
	UF : 0, UT : 6,		CONFIG : 'N U T, 0, 0, 0',
	X =  183.871  mm,	Y =   -494.426  mm,	Z =   -309.000  mm,
	W =  90.000 deg,	P =   0.000 deg,	R =   90.000 deg
};
P[3471]{
   GP1:
	UF : 0, UT : 6,		CONFIG : 'N U T, 0, 0, 0',
	X =  183.098  mm,	Y =   -494.562  mm,	Z =   -309.100  mm,
	W =  90.000 deg,	P =   0.000 deg,	R =   90.000 deg
};
P[3472]{
   GP1:
	UF : 0, UT : 6,		CONFIG : 'N U T, 0, 0, 0',
	X =  181.966  mm,	Y =   -495.196  mm,	Z =   -309.100  mm,
	W =  90.000 deg,	P =   0.000 deg,	R =   90.000 deg
};
P[3473]{
   GP1:
	UF : 0, UT : 6,		CONFIG : 'N U T, 0, 0, 0',
	X =  180.815  mm,	Y =   -495.373  mm,	Z =   -309.000  mm,
	W =  90.000 deg,	P =   0.000 deg,	R =   90.000 deg
};
P[3474]{
   GP1:
	UF : 0, UT : 6,		CONFIG : 'N U T, 0, 0, 0',
	X =  180.066  mm,	Y =   -495.745  mm,	Z =   -309.000  mm,
	W =  90.000 deg,	P =   0.000 deg,	R =   90.000 deg
};
P[3475]{
   GP1:
	UF : 0, UT : 6,		CONFIG : 'N U T, 0, 0, 0',
	X =  179.635  mm,	Y =   -496.505  mm,	Z =   -309.000  mm,
	W =  90.000 deg,	P =   0.000 deg,	R =   90.000 deg
};
P[3476]{
   GP1:
	UF : 0, UT : 6,		CONFIG : 'N U T, 0, 0, 0',
	X =  178.695  mm,	Y =   -497.074  mm,	Z =   -309.000  mm,
	W =  90.000 deg,	P =   0.000 deg,	R =   90.000 deg
};
P[3477]{
   GP1:
	UF : 0, UT : 6,		CONFIG : 'N U T, 0, 0, 0',
	X =  178.038  mm,	Y =   -497.441  mm,	Z =   -309.100  mm,
	W =  90.000 deg,	P =   0.000 deg,	R =   90.000 deg
};
P[3478]{
   GP1:
	UF : 0, UT : 6,		CONFIG : 'N U T, 0, 0, 0',
	X =  177.353  mm,	Y =   -497.812  mm,	Z =   -309.000  mm,
	W =  90.000 deg,	P =   0.000 deg,	R =   90.000 deg
};
P[3479]{
   GP1:
	UF : 0, UT : 6,		CONFIG : 'N U T, 0, 0, 0',
	X =  175.916  mm,	Y =   -498.217  mm,	Z =   -309.100  mm,
	W =  90.000 deg,	P =   0.000 deg,	R =   90.000 deg
};
P[3480]{
   GP1:
	UF : 0, UT : 6,		CONFIG : 'N U T, 0, 0, 0',
	X =  175.503  mm,	Y =   -499.150  mm,	Z =   -309.000  mm,
	W =  90.000 deg,	P =   0.000 deg,	R =   90.000 deg
};
P[3481]{
   GP1:
	UF : 0, UT : 6,		CONFIG : 'N U T, 0, 0, 0',
	X =  173.689  mm,	Y =   -499.966  mm,	Z =   -309.000  mm,
	W =  90.000 deg,	P =   0.000 deg,	R =   90.000 deg
};
P[3482]{
   GP1:
	UF : 0, UT : 6,		CONFIG : 'N U T, 0, 0, 0',
	X =  172.857  mm,	Y =   -500.307  mm,	Z =   -309.100  mm,
	W =  90.000 deg,	P =   0.000 deg,	R =   90.000 deg
};
P[3483]{
   GP1:
	UF : 0, UT : 6,		CONFIG : 'N U T, 0, 0, 0',
	X =  171.943  mm,	Y =   -500.753  mm,	Z =   -309.100  mm,
	W =  90.000 deg,	P =   0.000 deg,	R =   90.000 deg
};
P[3484]{
   GP1:
	UF : 0, UT : 6,		CONFIG : 'N U T, 0, 0, 0',
	X =  170.935  mm,	Y =   -501.394  mm,	Z =   -309.000  mm,
	W =  90.000 deg,	P =   0.000 deg,	R =   90.000 deg
};
P[3485]{
   GP1:
	UF : 0, UT : 6,		CONFIG : 'N U T, 0, 0, 0',
	X =  169.838  mm,	Y =   -501.932  mm,	Z =   -309.000  mm,
	W =  90.000 deg,	P =   0.000 deg,	R =   90.000 deg
};
P[3486]{
   GP1:
	UF : 0, UT : 6,		CONFIG : 'N U T, 0, 0, 0',
	X =  168.418  mm,	Y =   -502.881  mm,	Z =   -309.000  mm,
	W =  90.000 deg,	P =   0.000 deg,	R =   90.000 deg
};
P[3487]{
   GP1:
	UF : 0, UT : 6,		CONFIG : 'N U T, 0, 0, 0',
	X =  176.220  mm,	Y =   -516.018  mm,	Z =   -309.100  mm,
	W =  90.000 deg,	P =   0.000 deg,	R =   90.000 deg
};
P[3488]{
   GP1:
	UF : 0, UT : 6,		CONFIG : 'N U T, 0, 0, 0',
	X =  176.975  mm,	Y =   -515.678  mm,	Z =   -309.100  mm,
	W =  90.000 deg,	P =   0.000 deg,	R =   90.000 deg
};
P[3489]{
   GP1:
	UF : 0, UT : 6,		CONFIG : 'N U T, 0, 0, 0',
	X =  177.564  mm,	Y =   -514.505  mm,	Z =   -309.100  mm,
	W =  90.000 deg,	P =   0.000 deg,	R =   90.000 deg
};
P[3490]{
   GP1:
	UF : 0, UT : 6,		CONFIG : 'N U T, 0, 0, 0',
	X =  178.725  mm,	Y =   -514.348  mm,	Z =   -309.100  mm,
	W =  90.000 deg,	P =   0.000 deg,	R =   90.000 deg
};
P[3491]{
   GP1:
	UF : 0, UT : 6,		CONFIG : 'N U T, 0, 0, 0',
	X =  179.366  mm,	Y =   -513.759  mm,	Z =   -309.100  mm,
	W =  90.000 deg,	P =   0.000 deg,	R =   90.000 deg
};
P[3492]{
   GP1:
	UF : 0, UT : 6,		CONFIG : 'N U T, 0, 0, 0',
	X =  181.162  mm,	Y =   -512.893  mm,	Z =   -309.100  mm,
	W =  90.000 deg,	P =   0.000 deg,	R =   90.000 deg
};
P[3493]{
   GP1:
	UF : 0, UT : 6,		CONFIG : 'N U T, 0, 0, 0',
	X =  182.269  mm,	Y =   -512.296  mm,	Z =   -309.100  mm,
	W =  90.000 deg,	P =   0.000 deg,	R =   90.000 deg
};
P[3494]{
   GP1:
	UF : 0, UT : 6,		CONFIG : 'N U T, 0, 0, 0',
	X =  183.634  mm,	Y =   -511.349  mm,	Z =   -309.100  mm,
	W =  90.000 deg,	P =   0.000 deg,	R =   90.000 deg
};
P[3495]{
   GP1:
	UF : 0, UT : 6,		CONFIG : 'N U T, 0, 0, 0',
	X =  184.644  mm,	Y =   -510.368  mm,	Z =   -309.100  mm,
	W =  90.000 deg,	P =   0.000 deg,	R =   90.000 deg
};
P[3496]{
   GP1:
	UF : 0, UT : 6,		CONFIG : 'N U T, 0, 0, 0',
	X =  185.320  mm,	Y =   -510.390  mm,	Z =   -309.100  mm,
	W =  90.000 deg,	P =   0.000 deg,	R =   90.000 deg
};
P[3497]{
   GP1:
	UF : 0, UT : 6,		CONFIG : 'N U T, 0, 0, 0',
	X =  186.452  mm,	Y =   -510.175  mm,	Z =   -309.000  mm,
	W =  90.000 deg,	P =   0.000 deg,	R =   90.000 deg
};
P[3498]{
   GP1:
	UF : 0, UT : 6,		CONFIG : 'N U T, 0, 0, 0',
	X =  187.554  mm,	Y =   -509.641  mm,	Z =   -309.100  mm,
	W =  90.000 deg,	P =   0.000 deg,	R =   90.000 deg
};
P[3499]{
   GP1:
	UF : 0, UT : 6,		CONFIG : 'N U T, 0, 0, 0',
	X =  188.109  mm,	Y =   -508.896  mm,	Z =   -309.100  mm,
	W =  90.000 deg,	P =   0.000 deg,	R =   90.000 deg
};
P[3500]{
   GP1:
	UF : 0, UT : 6,		CONFIG : 'N U T, 0, 0, 0',
	X =  188.689  mm,	Y =   -508.140  mm,	Z =   -309.000  mm,
	W =  90.000 deg,	P =   0.000 deg,	R =   90.000 deg
};
P[3501]{
   GP1:
	UF : 0, UT : 6,		CONFIG : 'N U T, 0, 0, 0',
	X =  189.844  mm,	Y =   -507.796  mm,	Z =   -309.100  mm,
	W =  90.000 deg,	P =   0.000 deg,	R =   90.000 deg
};
P[3502]{
   GP1:
	UF : 0, UT : 6,		CONFIG : 'N U T, 0, 0, 0',
	X =  190.674  mm,	Y =   -507.286  mm,	Z =   -309.100  mm,
	W =  90.000 deg,	P =   0.000 deg,	R =   90.000 deg
};
P[3503]{
   GP1:
	UF : 0, UT : 6,		CONFIG : 'N U T, 0, 0, 0',
	X =  190.772  mm,	Y =   -506.803  mm,	Z =   -322.926  mm,
	W =  90.000 deg,	P =   0.000 deg,	R =   90.000 deg
};
P[3504]{
   GP1:
	UF : 0, UT : 6,		CONFIG : 'N U T, 0, 0, 0',
	X =  190.843  mm,	Y =   -506.926  mm,	Z =   -309.100  mm,
	W =  90.000 deg,	P =   0.000 deg,	R =   90.000 deg
};
P[3505]{
   GP1:
	UF : 0, UT : 6,		CONFIG : 'N U T, 0, 0, 0',
	X =  190.859  mm,	Y =   -506.954  mm,	Z =   -309.100  mm,
	W =  90.000 deg,	P =   0.000 deg,	R =   90.000 deg
};
P[3506]{
   GP1:
	UF : 0, UT : 6,		CONFIG : 'N U T, 0, 0, 0',
	X =  190.896  mm,	Y =   -507.018  mm,	Z =   -309.100  mm,
	W =  90.000 deg,	P =   0.000 deg,	R =   90.000 deg
};
P[3507]{
   GP1:
	UF : 0, UT : 6,		CONFIG : 'N U T, 0, 0, 0',
	X =  190.961  mm,	Y =   -507.131  mm,	Z =   -309.100  mm,
	W =  90.000 deg,	P =   0.000 deg,	R =   90.000 deg
};
P[3508]{
   GP1:
	UF : 0, UT : 6,		CONFIG : 'N U T, 0, 0, 0',
	X =  191.020  mm,	Y =   -507.233  mm,	Z =   -309.100  mm,
	W =  90.000 deg,	P =   0.000 deg,	R =   90.000 deg
};
P[3509]{
   GP1:
	UF : 0, UT : 6,		CONFIG : 'N U T, 0, 0, 0',
	X =  191.050  mm,	Y =   -507.285  mm,	Z =   -309.100  mm,
	W =  90.000 deg,	P =   0.000 deg,	R =   90.000 deg
};
P[3510]{
   GP1:
	UF : 0, UT : 6,		CONFIG : 'N U T, 0, 0, 0',
	X =  191.105  mm,	Y =   -507.380  mm,	Z =   -309.000  mm,
	W =  90.000 deg,	P =   0.000 deg,	R =   90.000 deg
};
P[3511]{
   GP1:
	UF : 0, UT : 6,		CONFIG : 'N U T, 0, 0, 0',
	X =  191.165  mm,	Y =   -507.484  mm,	Z =   -309.000  mm,
	W =  90.000 deg,	P =   0.000 deg,	R =   90.000 deg
};
P[3512]{
   GP1:
	UF : 0, UT : 6,		CONFIG : 'N U T, 0, 0, 0',
	X =  191.221  mm,	Y =   -507.581  mm,	Z =   -309.100  mm,
	W =  90.000 deg,	P =   0.000 deg,	R =   90.000 deg
};
P[3513]{
   GP1:
	UF : 0, UT : 6,		CONFIG : 'N U T, 0, 0, 0',
	X =  191.128  mm,	Y =   -507.318  mm,	Z =   -309.100  mm,
	W =  90.000 deg,	P =   0.000 deg,	R =   90.000 deg
};
P[3514]{
   GP1:
	UF : 0, UT : 6,		CONFIG : 'N U T, 0, 0, 0',
	X =  191.370  mm,	Y =   -507.108  mm,	Z =   -309.100  mm,
	W =  90.000 deg,	P =   0.000 deg,	R =   90.000 deg
};
P[3515]{
   GP1:
	UF : 0, UT : 6,		CONFIG : 'N U T, 0, 0, 0',
	X =  192.392  mm,	Y =   -506.475  mm,	Z =   -318.899  mm,
	W =  90.000 deg,	P =   0.000 deg,	R =   90.000 deg
};
P[3516]{
   GP1:
	UF : 0, UT : 6,		CONFIG : 'N U T, 0, 0, 0',
	X =  193.956  mm,	Y =   -505.600  mm,	Z =   -309.100  mm,
	W =  90.000 deg,	P =   0.000 deg,	R =   90.000 deg
};
P[3517]{
   GP1:
	UF : 0, UT : 6,		CONFIG : 'N U T, 0, 0, 0',
	X =  195.118  mm,	Y =   -504.754  mm,	Z =   -309.100  mm,
	W =  90.000 deg,	P =   0.000 deg,	R =   90.000 deg
};
P[3518]{
   GP1:
	UF : 0, UT : 6,		CONFIG : 'N U T, 0, 0, 0',
	X =  195.932  mm,	Y =   -504.090  mm,	Z =   -309.100  mm,
	W =  90.000 deg,	P =   0.000 deg,	R =   90.000 deg
};
P[3519]{
   GP1:
	UF : 0, UT : 6,		CONFIG : 'N U T, 0, 0, 0',
	X =  196.657  mm,	Y =   -503.969  mm,	Z =   -309.100  mm,
	W =  90.000 deg,	P =   0.000 deg,	R =   90.000 deg
};
P[3520]{
   GP1:
	UF : 0, UT : 6,		CONFIG : 'N U T, 0, 0, 0',
	X =  197.511  mm,	Y =   -503.502  mm,	Z =   -309.100  mm,
	W =  90.000 deg,	P =   0.000 deg,	R =   90.000 deg
};
P[3521]{
   GP1:
	UF : 0, UT : 6,		CONFIG : 'N U T, 0, 0, 0',
	X =  198.120  mm,	Y =   -503.154  mm,	Z =   -309.100  mm,
	W =  90.000 deg,	P =   0.000 deg,	R =   90.000 deg
};
P[3522]{
   GP1:
	UF : 0, UT : 6,		CONFIG : 'N U T, 0, 0, 0',
	X =  199.189  mm,	Y =   -502.492  mm,	Z =   -309.000  mm,
	W =  90.000 deg,	P =   0.000 deg,	R =   90.000 deg
};
P[3523]{
   GP1:
	UF : 0, UT : 6,		CONFIG : 'N U T, 0, 0, 0',
	X =  200.217  mm,	Y =   -502.061  mm,	Z =   -309.100  mm,
	W =  90.000 deg,	P =   0.000 deg,	R =   90.000 deg
};
P[3524]{
   GP1:
	UF : 0, UT : 6,		CONFIG : 'N U T, 0, 0, 0',
	X =  201.427  mm,	Y =   -501.402  mm,	Z =   -309.100  mm,
	W =  90.000 deg,	P =   0.000 deg,	R =   90.000 deg
};
P[3525]{
   GP1:
	UF : 0, UT : 6,		CONFIG : 'N U T, 0, 0, 0',
	X =  202.118  mm,	Y =   -501.068  mm,	Z =   -309.100  mm,
	W =  90.000 deg,	P =   0.000 deg,	R =   90.000 deg
};
P[3526]{
   GP1:
	UF : 0, UT : 6,		CONFIG : 'N U T, 0, 0, 0',
	X =  203.017  mm,	Y =   -500.557  mm,	Z =   -324.851  mm,
	W =  90.000 deg,	P =   0.000 deg,	R =   90.000 deg
};
P[3527]{
   GP1:
	UF : 0, UT : 6,		CONFIG : 'N U T, 0, 0, 0',
	X =  203.548  mm,	Y =   -499.609  mm,	Z =   -317.898  mm,
	W =  90.000 deg,	P =   0.000 deg,	R =   90.000 deg
};
P[3528]{
   GP1:
	UF : 0, UT : 6,		CONFIG : 'N U T, 0, 0, 0',
	X =  204.699  mm,	Y =   -499.393  mm,	Z =   -309.100  mm,
	W =  90.000 deg,	P =   0.000 deg,	R =   90.000 deg
};
P[3529]{
   GP1:
	UF : 0, UT : 6,		CONFIG : 'N U T, 0, 0, 0',
	X =  205.290  mm,	Y =   -498.939  mm,	Z =   -309.100  mm,
	W =  90.000 deg,	P =   0.000 deg,	R =   90.000 deg
};
P[3530]{
   GP1:
	UF : 0, UT : 6,		CONFIG : 'N U T, 0, 0, 0',
	X =  206.372  mm,	Y =   -498.018  mm,	Z =   -309.100  mm,
	W =  90.000 deg,	P =   0.000 deg,	R =   90.000 deg
};
P[3531]{
   GP1:
	UF : 0, UT : 6,		CONFIG : 'N U T, 0, 0, 0',
	X =  207.869  mm,	Y =   -498.001  mm,	Z =   -320.922  mm,
	W =  90.000 deg,	P =   0.000 deg,	R =   90.000 deg
};
P[3532]{
   GP1:
	UF : 0, UT : 6,		CONFIG : 'N U T, 0, 0, 0',
	X =  208.475  mm,	Y =   -496.578  mm,	Z =   -309.100  mm,
	W =  90.000 deg,	P =   0.000 deg,	R =   90.000 deg
};
P[3533]{
   GP1:
	UF : 0, UT : 6,		CONFIG : 'N U T, 0, 0, 0',
	X =  209.178  mm,	Y =   -496.381  mm,	Z =   -309.100  mm,
	W =  90.000 deg,	P =   0.000 deg,	R =   90.000 deg
};
P[3534]{
   GP1:
	UF : 0, UT : 6,		CONFIG : 'N U T, 0, 0, 0',
	X =  209.976  mm,	Y =   -496.397  mm,	Z =   -309.100  mm,
	W =  90.000 deg,	P =   0.000 deg,	R =   90.000 deg
};
P[3535]{
   GP1:
	UF : 0, UT : 6,		CONFIG : 'N U T, 0, 0, 0',
	X =  210.781  mm,	Y =   -495.904  mm,	Z =   -309.100  mm,
	W =  90.000 deg,	P =   0.000 deg,	R =   90.000 deg
};
P[3536]{
   GP1:
	UF : 0, UT : 6,		CONFIG : 'N U T, 0, 0, 0',
	X =  211.450  mm,	Y =   -495.368  mm,	Z =   -309.000  mm,
	W =  90.000 deg,	P =   0.000 deg,	R =   90.000 deg
};
P[3537]{
   GP1:
	UF : 0, UT : 6,		CONFIG : 'N U T, 0, 0, 0',
	X =  212.724  mm,	Y =   -494.989  mm,	Z =   -322.927  mm,
	W =  90.000 deg,	P =   0.000 deg,	R =   90.000 deg
};
P[3538]{
   GP1:
	UF : 0, UT : 6,		CONFIG : 'N U T, 0, 0, 0',
	X =  213.406  mm,	Y =   -494.335  mm,	Z =   -309.100  mm,
	W =  90.000 deg,	P =   0.000 deg,	R =   90.000 deg
};
P[3539]{
   GP1:
	UF : 0, UT : 6,		CONFIG : 'N U T, 0, 0, 0',
	X =  214.188  mm,	Y =   -494.207  mm,	Z =   -309.000  mm,
	W =  90.000 deg,	P =   0.000 deg,	R =   90.000 deg
};
P[3540]{
   GP1:
	UF : 0, UT : 6,		CONFIG : 'N U T, 0, 0, 0',
	X =  215.596  mm,	Y =   -492.702  mm,	Z =   -309.100  mm,
	W =  90.000 deg,	P =   0.000 deg,	R =   90.000 deg
};
P[3541]{
   GP1:
	UF : 0, UT : 6,		CONFIG : 'N U T, 0, 0, 0',
	X =  216.619  mm,	Y =   -492.598  mm,	Z =   -309.100  mm,
	W =  90.000 deg,	P =   0.000 deg,	R =   90.000 deg
};
P[3542]{
   GP1:
	UF : 0, UT : 6,		CONFIG : 'N U T, 0, 0, 0',
	X =  217.216  mm,	Y =   -492.151  mm,	Z =   -309.100  mm,
	W =  90.000 deg,	P =   0.000 deg,	R =   90.000 deg
};
P[3543]{
   GP1:
	UF : 0, UT : 6,		CONFIG : 'N U T, 0, 0, 0',
	X =  218.313  mm,	Y =   -491.828  mm,	Z =   -309.000  mm,
	W =  90.000 deg,	P =   0.000 deg,	R =   90.000 deg
};
P[3544]{
   GP1:
	UF : 0, UT : 6,		CONFIG : 'N U T, 0, 0, 0',
	X =  219.143  mm,	Y =   -491.501  mm,	Z =   -309.100  mm,
	W =  90.000 deg,	P =   0.000 deg,	R =   90.000 deg
};
P[3545]{
   GP1:
	UF : 0, UT : 6,		CONFIG : 'N U T, 0, 0, 0',
	X =  219.812  mm,	Y =   -490.234  mm,	Z =   -309.100  mm,
	W =  90.000 deg,	P =   0.000 deg,	R =   90.000 deg
};
P[3546]{
   GP1:
	UF : 0, UT : 6,		CONFIG : 'N U T, 0, 0, 0',
	X =  220.608  mm,	Y =   -489.974  mm,	Z =   -309.100  mm,
	W =  90.000 deg,	P =   0.000 deg,	R =   90.000 deg
};
P[3547]{
   GP1:
	UF : 0, UT : 6,		CONFIG : 'N U T, 0, 0, 0',
	X =  221.733  mm,	Y =   -489.622  mm,	Z =   -325.004  mm,
	W =  90.000 deg,	P =   0.000 deg,	R =   90.000 deg
};
P[3548]{
   GP1:
	UF : 0, UT : 6,		CONFIG : 'N U T, 0, 0, 0',
	X =  222.481  mm,	Y =   -489.503  mm,	Z =   -309.100  mm,
	W =  90.000 deg,	P =   0.000 deg,	R =   90.000 deg
};
P[3549]{
   GP1:
	UF : 0, UT : 6,		CONFIG : 'N U T, 0, 0, 0',
	X =  223.355  mm,	Y =   -488.417  mm,	Z =   -309.100  mm,
	W =  90.000 deg,	P =   0.000 deg,	R =   90.000 deg
};
P[3550]{
   GP1:
	UF : 0, UT : 6,		CONFIG : 'N U T, 0, 0, 0',
	X =  224.448  mm,	Y =   -488.318  mm,	Z =   -309.100  mm,
	W =  90.000 deg,	P =   0.000 deg,	R =   90.000 deg
};
P[3551]{
   GP1:
	UF : 0, UT : 6,		CONFIG : 'N U T, 0, 0, 0',
	X =  225.418  mm,	Y =   -487.694  mm,	Z =   -309.000  mm,
	W =  90.000 deg,	P =   0.000 deg,	R =   90.000 deg
};
P[3552]{
   GP1:
	UF : 0, UT : 6,		CONFIG : 'N U T, 0, 0, 0',
	X =  226.290  mm,	Y =   -486.879  mm,	Z =   -319.186  mm,
	W =  90.000 deg,	P =   0.000 deg,	R =   90.000 deg
};
P[3553]{
   GP1:
	UF : 0, UT : 6,		CONFIG : 'N U T, 0, 0, 0',
	X =  227.233  mm,	Y =   -486.363  mm,	Z =   -321.230  mm,
	W =  90.000 deg,	P =   0.000 deg,	R =   90.000 deg
};
P[3554]{
   GP1:
	UF : 0, UT : 6,		CONFIG : 'N U T, 0, 0, 0',
	X =  228.080  mm,	Y =   -486.020  mm,	Z =   -309.100  mm,
	W =  90.000 deg,	P =   0.000 deg,	R =   90.000 deg
};
P[3555]{
   GP1:
	UF : 0, UT : 6,		CONFIG : 'N U T, 0, 0, 0',
	X =  228.515  mm,	Y =   -485.138  mm,	Z =   -309.949  mm,
	W =  90.000 deg,	P =   0.000 deg,	R =   90.000 deg
};
P[3556]{
   GP1:
	UF : 0, UT : 6,		CONFIG : 'N U T, 0, 0, 0',
	X =  229.534  mm,	Y =   -485.508  mm,	Z =   -309.100  mm,
	W =  90.000 deg,	P =   0.000 deg,	R =   90.000 deg
};
P[3557]{
   GP1:
	UF : 0, UT : 6,		CONFIG : 'N U T, 0, 0, 0',
	X =  230.006  mm,	Y =   -484.509  mm,	Z =   -309.000  mm,
	W =  90.000 deg,	P =   0.000 deg,	R =   90.000 deg
};
P[3558]{
   GP1:
	UF : 0, UT : 6,		CONFIG : 'N U T, 0, 0, 0',
	X =  231.202  mm,	Y =   -484.445  mm,	Z =   -309.100  mm,
	W =  90.000 deg,	P =   0.000 deg,	R =   90.000 deg
};
P[3559]{
   GP1:
	UF : 0, UT : 6,		CONFIG : 'N U T, 0, 0, 0',
	X =  231.350  mm,	Y =   -483.376  mm,	Z =   -309.100  mm,
	W =  90.000 deg,	P =   0.000 deg,	R =   90.000 deg
};
P[3560]{
   GP1:
	UF : 0, UT : 6,		CONFIG : 'N U T, 0, 0, 0',
	X =  232.545  mm,	Y =   -483.626  mm,	Z =   -309.100  mm,
	W =  90.000 deg,	P =   0.000 deg,	R =   90.000 deg
};
P[3561]{
   GP1:
	UF : 0, UT : 6,		CONFIG : 'N U T, 0, 0, 0',
	X =  234.135  mm,	Y =   -482.125  mm,	Z =   -309.100  mm,
	W =  90.000 deg,	P =   0.000 deg,	R =   90.000 deg
};
P[3562]{
   GP1:
	UF : 0, UT : 6,		CONFIG : 'N U T, 0, 0, 0',
	X =  234.868  mm,	Y =   -481.999  mm,	Z =   -309.000  mm,
	W =  90.000 deg,	P =   0.000 deg,	R =   90.000 deg
};
P[3563]{
   GP1:
	UF : 0, UT : 6,		CONFIG : 'N U T, 0, 0, 0',
	X =  235.666  mm,	Y =   -481.320  mm,	Z =   -309.100  mm,
	W =  90.000 deg,	P =   0.000 deg,	R =   90.000 deg
};
P[3564]{
   GP1:
	UF : 0, UT : 6,		CONFIG : 'N U T, 0, 0, 0',
	X =  237.549  mm,	Y =   -480.558  mm,	Z =   -309.100  mm,
	W =  90.000 deg,	P =   0.000 deg,	R =   90.000 deg
};
P[3565]{
   GP1:
	UF : 0, UT : 6,		CONFIG : 'N U T, 0, 0, 0',
	X =  238.299  mm,	Y =   -479.938  mm,	Z =   -323.464  mm,
	W =  90.000 deg,	P =   0.000 deg,	R =   90.000 deg
};
P[3566]{
   GP1:
	UF : 0, UT : 6,		CONFIG : 'N U T, 0, 0, 0',
	X =  239.183  mm,	Y =   -479.481  mm,	Z =   -309.100  mm,
	W =  90.000 deg,	P =   0.000 deg,	R =   90.000 deg
};
P[3567]{
   GP1:
	UF : 0, UT : 6,		CONFIG : 'N U T, 0, 0, 0',
	X =  239.933  mm,	Y =   -478.853  mm,	Z =   -326.022  mm,
	W =  90.000 deg,	P =   0.000 deg,	R =   90.000 deg
};
P[3568]{
   GP1:
	UF : 0, UT : 6,		CONFIG : 'N U T, 0, 0, 0',
	X =  240.878  mm,	Y =   -478.509  mm,	Z =   -309.100  mm,
	W =  90.000 deg,	P =   0.000 deg,	R =   90.000 deg
};
P[3569]{
   GP1:
	UF : 0, UT : 6,		CONFIG : 'N U T, 0, 0, 0',
	X =  242.422  mm,	Y =   -477.447  mm,	Z =   -309.100  mm,
	W =  90.000 deg,	P =   0.000 deg,	R =   90.000 deg
};
P[3570]{
   GP1:
	UF : 0, UT : 6,		CONFIG : 'N U T, 0, 0, 0',
	X =  243.065  mm,	Y =   -477.429  mm,	Z =   -309.100  mm,
	W =  90.000 deg,	P =   0.000 deg,	R =   90.000 deg
};
P[3571]{
   GP1:
	UF : 0, UT : 6,		CONFIG : 'N U T, 0, 0, 0',
	X =  243.288  mm,	Y =   -476.895  mm,	Z =   -309.100  mm,
	W =  90.000 deg,	P =   0.000 deg,	R =   90.000 deg
};
P[3572]{
   GP1:
	UF : 0, UT : 6,		CONFIG : 'N U T, 0, 0, 0',
	X =  244.503  mm,	Y =   -476.316  mm,	Z =   -309.100  mm,
	W =  90.000 deg,	P =   0.000 deg,	R =   90.000 deg
};
P[3573]{
   GP1:
	UF : 0, UT : 6,		CONFIG : 'N U T, 0, 0, 0',
	X =  245.241  mm,	Y =   -475.676  mm,	Z =   -309.100  mm,
	W =  90.000 deg,	P =   0.000 deg,	R =   90.000 deg
};
P[3574]{
   GP1:
	UF : 0, UT : 6,		CONFIG : 'N U T, 0, 0, 0',
	X =  246.209  mm,	Y =   -475.442  mm,	Z =   -321.566  mm,
	W =  90.000 deg,	P =   0.000 deg,	R =   90.000 deg
};
P[3575]{
   GP1:
	UF : 0, UT : 6,		CONFIG : 'N U T, 0, 0, 0',
